FUNCTION_BLOCK "Ponsel_mesure"   // FB107, SCL
{ S7_Optimized_Access := 'TRUE' }
VERSION : 0.1
   VAR_INPUT
      mb_addr : UInt;
      minimum_measurement_interval : Time := T#1M;
      compensate_enable : Bool;
      compensate : Array[1..2] of Real;
   END_VAR
   VAR_OUTPUT
      Measurement_ok : Bool;
   END_VAR
   VAR_IN_OUT
      mb_query : "mb_query";
      start_measurement : Bool;
   END_VAR
   VAR
      sb : "mb_station_block_udt";
      QueryCnt : UDInt;
      data1 : Struct
         value : Array[0..4] of Real;
         compensate_temperature : Real;
         compensate : Array[1..2] of Real;
         _ : Word;
         status : Array[0..4] of Struct
            x08_StmGamme0 : Bool;
            x09_StmGamme1 : Bool;
            x10_StmGamme2 : Bool;
            x11 : Bool;
            x12 : Bool;
            x13 : Bool;
            x14 : Bool;
            x15 : Bool;
            x00_Stm0 : Bool;
            x01_Stm1 : Bool;
            x02_Stm2 : Bool;
            x03_StmTemp : Bool;   // At least one parameter coefficient uses a temporary calibration standard (configuration during calibration)
            x04_StmHF : Bool;   // At least one parameter coefficient is outside calibration limits
            x05_StmCU : Bool;   // All parameter coefficients use default coefficient
            x06_StmHIST : Bool;   // All parameter coefficients use history coefficient
            x07_StmME : Bool;   // Dry weight is missing in at least one parameter coefficient (measurement under way)
         END_STRUCT;
         Compensates_3 : Real;
      END_STRUCT;
      data2 : Struct
         Description : String[30];
         serial_number : String[32];   // (addr 0x0D10)
         Software_version : Word;   // Heavy Weight: Major version and Light Weight: Minor Version.
         Hardware_version : Word;   // Heavy Weight: Major version and Light Weight: Minor Version.
      END_STRUCT;
      api : Struct
         idle : Bool;
         wait : Bool;
         interval : Time;
      END_STRUCT;
      _ : Bool;   // Internal variables bellow.
      state : Int;
      "timer" : TON_TIME;
      timer_in : Bool;
      timer_q : Bool;
      first_scan : Bool := TRUE;
      wait_time : UInt;
   END_VAR
   VAR_TEMP
      "word" : Word;
      c : Int;
      error : Bool;
      tIdle : Bool;
      pt : Time;
   END_VAR
BEGIN
   // Aqualabo - Ponsel mesure
   // Dissolved oxygen (OPTOD), Conductivity (C4E, CTZ), pH_Redox, Turbi    
   // 
   // - Warning: For the oxygen sensor each pull for sensor measurement,
   //   will use of the available life span. Please set the measurement
   //   interval to appropriate value.
   // - Continuous assign true to start_measurement, to continuous do
   //   meassurements. #minimum_measurement_interval wil still restrict
   //   the interval time.
   // - https://en.aqualabo.fr/userfiles/doc/User%20Manual%20Oxygen%20Optical%20digital%20sensor%20OPTOD.pdf

   "mb_station_block_header"(sb := #sb,
                             mb_query := #mb_query);
   #mb_query.mb_addr := #mb_addr;
   #mb_query.mode := #mb_query.c.read.holding_reg;

   #"timer"(IN := #timer_in,
          PT := #"timer".PT,
          Q => #timer_q);
   #timer_in := false;

   IF #sb.out.communication_error THEN // If communication error
       #state := 0;
       #Measurement_ok := false;
       #timer_in := true;  // Continue run the timer.
   ELSE
       CASE #state OF
           1:  // Compensate: Salinity, barometric pressure, temperature, etc.
               IF #compensate_enable THEN
                   #mb_query(mode := #mb_query.c.write.holding_reg,
                             data_addr := 16#5f,
                             data_ptr := #compensate);
                   #state += BOOL_TO_INT(#mb_query.Done);
               ELSE
                   #state += 1;
               END_IF;
           2:  // Read wait-time (Used later in state 4)
               #mb_query(data_addr := 16#A4,
                         data_ptr := #wait_time);
               #state += BOOL_TO_INT(#mb_query.Done);
           3:  // Start all meassurements.
               #"word" := 16#0f;
               #mb_query(mode := #mb_query.c.write.holding_reg,
                         data_addr := 16#01,
                         data_ptr := #"word");
               #state += BOOL_TO_INT(#mb_query.Done);
           4:  // Timer (Wait while sensor is obtaining measurements)
               #timer_in := true;
               PRESET_TIMER(TIMER := #"timer",
                            PT := MAX(IN1 := T_CONV(#wait_time),
                                      IN2 := T#1s)); // No less then 1s.
               #state += BOOL_TO_INT(#timer_q);
           5:  // Get data.
               #mb_query(data_addr := 16#0053,
                         data_ptr := #data1);
               // All measurements ok ?
               FOR #c := 0 TO 4 DO
                   #error := #error
                   OR #data1.status[#c].x00_Stm0
                   OR #data1.status[#c].x01_Stm1
                   OR #data1.status[#c].x02_Stm2;
               END_FOR;
               #Measurement_ok := NOT #error;
               IF #mb_query.Done THEN
                   // #start_measurement need to be assigned
                   // true again to start a new messurement.
                   #start_measurement := false;
                   #state := 0;
                   #QueryCnt += 1;
               END_IF;
           ELSE
               #tIdle := true;
               #timer_in := true;
               #pt := SEL(G := #api.interval = T#0s,
                          IN0 := #api.interval,
                          IN1 := #minimum_measurement_interval);
               PRESET_TIMER(PT := #pt,
                            TIMER := #"timer");

               #state := BOOL_TO_INT
               (NOT #api.wait AND // #api.wait may be set by other
                // function blocks to  halt the messurements.
                #start_measurement AND (
                (* *)#timer_q // Interval controlled
                (* *)OR #first_scan)); // At statup a messurement
               // is done as fast as possible.
       END_CASE;
   END_IF;
   // #wait is a API, for other blocks to stop the messurements,
   // #idle tells other blocks that no messurement is in progress.


   IF #sb.out.communication_error
       OR #api.idle AND NOT #api.wait
   THEN
       // Description, Serial number, sw and hw version.
       #mb_query(data_addr := 3327,
                 data_ptr := #data2);
   END_IF;

   "mb_station_block_footer"(sb := #sb,
                             mb_query := #mb_query);

   #api.idle := #tIdle;
   #api.wait := false;
   #api.interval := T#0s;
   #first_scan := false;

   (* 
   Units:
   ---------------
   value0: Temperature
                         value1:                    value2:                    value3:       
   OPTOD (oxygen)    :   Oxygen [%Sat]              Oxygen [mg/l]              Oxygen [ppm]
   Turbi             :   Nephelo turbidity [NTU]    Nephelo turbidity [FNU]    TU turbidity [mg/L]
   pH_Redox          :   pH                         Redox [mV]
   conductivity_C4E  :   Conductivity C4E [uS/cm]   Salinity [ppt]             TDS - Kcl [ppm]
   Conductivity_CTZ  :   Conductivity CTZ [mS/cm]   Salinity [g/Kg]            Conductivity CTZ [mS/cm] 
                                                                               without temperature compensation                                                                  
   OPTOD: (Dissolved oxygen)
   Compensates[1]: Atmospheric pressure [hPa], default 1013 hPa
   Compensates[2]: Salinity [ppt], default 0 ppt


   Wiring: 
   Red     Wiring diagram V+
   black   Wiring diagram V-
   Green   B+ RS-485  (Siemens A)
   White   A- RS-485  (Siemens B)
   Blue    SDI-12

   Default settings:
   Buad: 9600
   Parity: none
   Modbus address: 10


   StmX:
   000: Measurement OK
   001: Measurement OK, but out of specifications
   010: Measurement OK with INFO 1 (See datasheet)
   011: Measurement OK with INFO 2 (See datasheet)
   100: Measurement impossible, out of specifications
   101: Measurement impossible with INFO 3 (See datasheet)
   110: Measurement impossible with INFO 4 (See datasheet)
   111: measurement under way (not yet available)

   StmGamme:       
   001: measurement used range 1
   010: measurement used range 2
   011: measurement used range 3
   100: measurement used range 4

   *)
END_FUNCTION_BLOCK

// folder: Library/Modbus/Station blocks/sb tested/Siemens

FUNCTION_BLOCK "siemens_PAC3200"   // FB8, SCL
{ S7_Optimized_Access := 'TRUE' }
VERSION : 0.1
   VAR_INPUT
      mb_addr : USInt := 1;
   END_VAR
   VAR_IN_OUT
      mb_query : "mb_query";
   END_VAR
   VAR
      sb : "mb_station_block_udt";
      read1 : Struct
         voltage_L_n : Array[1..3] of Real;
         "voltage _L_L" : Array[1..3] of Real;   // 1:Va-b, 2:Vb-c, 3:Vc-a,
         current : Array[1..3] of Real;
         apparent_power : Array[1..3] of Real;
         active_power : Array[1..3] of Real;
         reactive_power : Array[1..3] of Real;
         power_factor : Array[1..3] of Real;
         THD_R_voltage : Array[1..3] of Real;
      END_STRUCT;
      read2 : Struct
         frequency : Real;   // unit: hz
         avg_voltage_Vph_n : Real;   // unit: V
         avg_voltage_Vph_ph : Real;   // unit: V
         avg_current : Real;   // unit: A
         total_apparent_power : Real;   // unit: VA
         total_active_power : Real;   // unit: W
      END_STRUCT;
   END_VAR
BEGIN
   // Siemens - PAC3200 - Power meter
   // 
   // Manual: 3.9.3, page 40

   "mb_station_block_header"(sb := #sb, mb_query := #mb_query);
   #mb_query.mb_addr := #mb_addr; // Device address.

   // Two queries, reading one section of holding registers each.
   #mb_query.mode := #mb_query.c.read.holding_reg;
   #mb_query(data_addr := 1, data_ptr := #read1);
   #mb_query(data_addr := 55, data_ptr := #read2);
   // - Each query reading one section of holding registers.
   // - Data length is automatically calculated for holding and input regisers.

   "mb_station_block_footer"(sb := #sb, mb_query := #mb_query);
END_FUNCTION_BLOCK

// folder: Library/Modbus/Station blocks/sb tested/zz Internal special

FUNCTION_BLOCK "temeratur_transmitter"   // FB2, SCL
{ S7_Optimized_Access := 'TRUE' }
VERSION : 0.1
   VAR_OUTPUT
      Temperatur : Real;
   END_VAR
   VAR_IN_OUT
      mb_query : "mb_query";
   END_VAR
   VAR
      sb : "mb_station_block_udt";
   END_VAR
   VAR_TEMP
      tmp : Int;
   END_VAR
BEGIN
   // Temperatur transmitter.

   "mb_station_block_header"(sb := #sb, mb_query := #mb_query);

   #mb_query(mb_addr := 1,
             mode := #mb_query.c.read.holding_reg,
             data_addr := 0,
             data_ptr := #tmp);

   IF #mb_query.Done THEN
       #Temperatur := REAL_TO_INT(#tmp) / 10;
   END_IF;

   "mb_station_block_footer"(sb := #sb, mb_query := #mb_query);
END_FUNCTION_BLOCK

// folder: Library/Modbus/Station blocks/sb untested

FUNCTION_BLOCK "Allen_bradley_power_flex_4"   // FB16, SCL
{ S7_Optimized_Access := 'TRUE' }
VERSION : 0.1
   VAR_INPUT
      mb_addr : USInt;
      ref : Real;
      reverse : Bool;
      reset : Bool;
   END_VAR
   VAR_OUTPUT
      Output_Frequency : Real;
      Output_Current : Real;
      DC_Bus_Voltage : Real;
      Output_Voltage : Real;
   END_VAR
   VAR_IN_OUT
      mb_query : "mb_query";
   END_VAR
   VAR
      sb : "mb_station_block_udt";
      read : Struct
         stat : Struct
            x08_At_Reference : Bool;
            x09_Reference_Controlled_by_Comm : Bool;
            x10_Operation_Cmd_Controlled_by_Comm : Bool;
            x11_Parameters_have_been_locked : Bool;
            x12_Digital_Input_1_Status : Bool;
            x13_Digital_Input_2_Status : Bool;
            x14 : Bool;
            x15 : Bool;
            "x00_Ready," : Bool;
            x01_Running : Bool;
            x02_cmd_Forward : Bool;
            x03_Rotating_Forward : Bool;
            x04_Accelerating : Bool;
            "x05_Decelerating," : Bool;
            x06_Alarm : Bool;
            x07_Faulted : Bool;
         END_STRUCT;
         error_code : UInt;
         ref_feedback : UInt;
         Output_Frequency : UInt;
         Output_Current : UInt;
         DC_Bus_Voltage : UInt;
         Output_Voltage : UInt;
      END_STRUCT;
      write : Struct
         cmd : Struct
            "x08_Accel Rate 1" : Bool := TRUE;
            "x09_Accel Rate 2" : Bool;
            "x10_Decel Rate 1" : Bool := TRUE;
            "x11_Decel Rate 2" : Bool;
            x12_Freq_Source_b0 : Bool := TRUE;
            x13_Freq_Source_b1 : Bool := TRUE;
            x14_Freq_Source_b2 : Bool;
            x15 : Bool;
            x00_Stop : Bool;
            x01_Start : Bool;
            x02_Jog : Bool;
            x03_Clear_Faults : Bool;
            x04_Forward : Bool;
            x05_Reverse : Bool;
            x06 : Bool;
            x07 : Bool;
         END_STRUCT;
         ref : UInt;
      END_STRUCT;
   END_VAR
BEGIN
   // Allen Bradley - Power Flex 4 - Compact AC Drive
   //
   // http://ab.rockwellautomation.com/Drives/PowerFlex-4
   // Web: https://plc-hmi-scadas.com/gallery/PowerFlex4ModBusAddressing.pdf

   "mb_station_block_header"(sb := #sb,
                             mb_query := #mb_query);
   #mb_query.mb_addr := #mb_addr;

   #write.ref := REAL_TO_UINT(#ref * 10);
   #write.cmd.x00_Stop := #ref = 0;
   #write.cmd.x01_Start := #ref <> 0;
   #write.cmd.x03_Clear_Faults := #reset;
   #write.cmd.x04_Forward := NOT #reverse;
   #write.cmd.x05_Reverse := #reverse;

   #mb_query.mode := #mb_query.c.write.single_holding_reg;
   #mb_query(data_addr := 8192,
             data_ptr := #write.cmd);
   #mb_query(data_addr := 8193,
             data_ptr := #write.ref);

   #mb_query.mode := #mb_query.c.read.holding_reg;
   #mb_query(data_addr := 8448,
             data_ptr := #read);
   #Output_Frequency := UINT_TO_REAL(#read.Output_Frequency) / 10;
   #Output_Current := UINT_TO_REAL(#read.Output_Current) / 100;
   #DC_Bus_Voltage := UINT_TO_REAL(#read.DC_Bus_Voltage) / 10;
   #Output_Voltage := UINT_TO_REAL(#read.Output_Voltage) / 10;

   "mb_station_block_footer"(sb := #sb,
                             mb_query := #mb_query);

   (* Error codes: (read.error_codes)
   0 - No Fault
   2 - Auxilary Input
   3 - Power Loss
   4 - Undervoltage
   5 - Overvoltage
   6 - Motor Stalled
   7 - Motor Overload
   8 - Heatsink Overtemperature
   12 - HW Overcurrent (300%)
   13 - Ground Fault
   29 - Analog Input Loss
   33 - Auto Restart Tries
   38 - Phase U to Ground Short
   39 - Phase V to Ground Short
   40 - Phase W to Ground Short
   41 - Phase U/V Short
   42 - Phase U/W Short
   43 - Phase V/W Short
   63 - Software Overcurrent
   64 - Drive Overload
   70 - Power Unit Fail
   80 - AutoTune Fail
   81 - Communication Loss
   100 - Parameter Checksum Error
   122 - I/O Board Fail         
   *)
END_FUNCTION_BLOCK

FUNCTION_BLOCK "Auma_valve"   // FB17, SCL
{ S7_Optimized_Access := 'TRUE' }
VERSION : 0.1
   VAR_INPUT
      mb_addr : UInt;
   END_VAR
   VAR_IN_OUT
      mb_query : "mb_query";
   END_VAR
   VAR
      sb : "mb_station_block_udt";
      read : Struct
         status : Struct
            torque_sw_closed : Bool;
            torque_sw_open : Bool;
            limit_sw_closed : Bool;
            limit_sw_open : Bool;
            sel_sw_local : Bool;
            sel_sw_remote : Bool;
            phase_fault : Bool;
            therminal_fault : Bool;
            falt : Bool;
            warning : Bool;
            running_close : Bool;
            running_open : Bool;
            not_ready_remote : Bool;
            setpoint_reached : Bool;
            end_p_clossed : Bool;
            end_p_open : Bool;
         END_STRUCT;
         "Actual position" : UInt;
      END_STRUCT;
      write : Struct
         cmd : Struct
            byte_2 : Byte;
            open : Bool;
            close : Bool;
            use_setpoint : Bool;
            reset : Bool;
            b4 : Bool;
            b5 : Bool;
            b6 : Bool;
            b7 : Bool;
         END_STRUCT;
         setpoint : UInt;
      END_STRUCT;
   END_VAR
BEGIN
   // Auma actuator controls
   // AC 01.2/ACExC 01.2 Modbus RTU
   //
   // http://www1.auma.com/uploads/media/sp_import2/handbuecher/
   // steuerungen/hb_ac2_modbus_geraeteintegration_en.pdf

   "mb_station_block_header"(sb := #sb, mb_query := #mb_query);
   #mb_query.mb_addr := #mb_addr;

   #mb_query(mode := #mb_query.c.read.input_reg,
             data_addr := 16#03E8,
             data_ptr := #read); // p.10

   #mb_query(mode := #mb_query.c.write.holding_reg,
             data_addr := 16#03E8,
             data_ptr := #write); // p.29

   "mb_station_block_footer"(sb := #sb, mb_query := #mb_query);

   (*
   - Each query reading one section of holding registers.
   - Data length is automatically calculated for holding 
     and input regisers.
   *)
END_FUNCTION_BLOCK

FUNCTION_BLOCK "Automatic_systems_AS1320"   // FB18, SCL
{ S7_Optimized_Access := 'TRUE' }
VERSION : 0.1
   VAR_INPUT
      mb_addr : UInt;
   END_VAR
   VAR_IN_OUT
      mb_query : "mb_query";
   END_VAR
   VAR
      sb : "mb_station_block_udt";
      read1 : Struct
         input : Word;
         input_3 : Word;
         output : Word;
         analog_in : Word;
         analog_out : Word;
         z2 : Array[1..4] of Word;
         temperature : Int;
         counter_1 : UDInt;
         counter_2 : UDInt;
         z : Array[1..3] of Word;
         state : Struct
            x08_blocked_closed : Bool;
            x09 : Bool;
            x10 : Bool;
            x11 : Bool;
            x12 : Bool;
            x13 : Bool;
            x14 : Bool;
            x15 : Bool;
            x00 : Bool;
            x01 : Bool;
            x02_open : Bool;
            x03_opening : Bool;
            x04_closed : Bool;
            x05_closing : Bool;
            x06_stop : Bool;
            x07_blocked_open : Bool;
         END_STRUCT;
      END_STRUCT;
      read2 : Struct
         PRDSTD : String[6];
         BL_xxx : String[6];
         "Type" : UInt;
         Change : UInt;
      END_STRUCT;
      write1 : Struct
         x08 : Bool;
         x09 : Bool;
         x10 : Bool;
         x11 : Bool;
         x12 : Bool;
         x13 : Bool;
         x14 : Bool;
         x15 : Bool;
         x00_open : Bool;
         x01_close : Bool;
         x02_block_open : Bool;
         x03_block_close : Bool;
         x04_stop : Bool;
         x05_reader_command_direction_a : Bool;
         x06_reader_command_direction_b : Bool;
         x07_reset_block : Bool;
      END_STRUCT;
      start_setup : Bool;
      write2 : Struct
         PS1_function : UInt;
         PS2_function : UInt;
         Positioning : UInt;
         barrier_type : UInt;
         arm_length : UInt;
         arm_type : UInt;
         power_fail_OP : UInt;
         exploitation : UInt;
      END_STRUCT;
      crank : Bool;
   END_VAR
BEGIN
   // Automatic systems - AS1320
   // http://www.visionbr.com.br/arquivo-produtos/20110823_92924_as1320-mt-en-16.pdf
   // Revision no: AS1320-prog 6.x-MT-FR-16 - 2009-11-10 

   "mb_station_block_header"(sb := #sb, mb_query := #mb_query);
   #mb_query.mb_addr := #mb_addr;

   #mb_query.mode := #mb_query.c.read.holding_reg;
   #mb_query(data_addr := 16#39, data_ptr := #read1);
   // #mb_query(data_addr := 16#00, data_ptr := #read3);
   // A micro switch at opening for the crank.
   #crank := #read1.input.%X14; 

   #mb_query.mode := #mb_query.c.write.holding_reg;
   #mb_query(data_addr := 16#12C, data_ptr := #write1);
   IF #start_setup THEN
       #mb_query(data_addr := 16#64, data_ptr := #write2);
       #start_setup := NOT #mb_query.Done;
   END_IF;

   "mb_station_block_footer"(sb := #sb, mb_query := #mb_query);
END_FUNCTION_BLOCK

FUNCTION_BLOCK "Belimo_vav_Compact_mod"   // FB19, SCL
{ S7_Optimized_Access := 'TRUE' }
VERSION : 0.1
   VAR_INPUT
      mb_addr : UInt;
      sp : Real;   // setpoint
      bus_fail_position : Real;
   END_VAR
   VAR_OUTPUT
      pos_feedback : Real;
   END_VAR
   VAR_IN_OUT
      mb_query : "mb_query";
   END_VAR
   VAR
      sb : "mb_station_block_udt";
      read : Struct
         position : Int;
      END_STRUCT;
      write1 : Struct
         setpoint : Int;
      END_STRUCT;
      write2 : Struct
         bus_fail_position : Int;
      END_STRUCT;
   END_VAR
BEGIN
   // Belimo - VAV-Compact MOD 
   // LMV-D3-MOD 5  Nm 2   W 4 VA (max. 5 A @ 5 ms) Approx. 500 g
   // NMV-D3-MOD 10 Nm 3.5 W 6 VA (max. 5 A @ 5 ms) Approx. 700 g
   // https://www.micromatic.no/globalassets/inriver/
   // resources/ko1070_0_5_1.pdf

   "mb_station_block_header"(sb := #sb, mb_query := #mb_query);
   #mb_query.mb_addr := #mb_addr;

   #mb_query.mode := #mb_query.c.read.holding_reg;
   #mb_query(data_addr := 4, data_ptr := #read);
   #pos_feedback := INT_TO_REAL(#read.position) * 0.01;

   #mb_query.mode := #mb_query.c.write.holding_reg;
   #write1.setpoint := REAL_TO_INT(#sp) * 100;
   #mb_query(data_addr := 0, data_ptr := #write1);
   #write2.bus_fail_position := REAL_TO_INT(#bus_fail_position) * 100;
   #mb_query(data_addr := 108, data_ptr := #write2);

   "mb_station_block_footer"(sb := #sb, mb_query := #mb_query);

   (*
   Bus fail position:
   0 Last setpoint (no bus monitoring)
   1 Fast close if time is exceeded
   2 Fast open if time is exceeded 
   *)
END_FUNCTION_BLOCK

FUNCTION_BLOCK "Binmaster_mnu_ultrasonic_sensor"   // FB20, SCL
{ S7_Optimized_Access := 'TRUE' }
VERSION : 0.1
   VAR_INPUT
      mb_addr : UInt;
   END_VAR
   VAR_IN_OUT
      mb_query : "mb_query";
   END_VAR
   VAR
      sb : "mb_station_block_udt";
      data : Struct
         "Model Type" : UInt;
         Raw_Distance_Level : UInt;   // [mm]
         _ : UInt;
         Temperature : Int;
         Calculated : DInt;
         __ : DWord;
         "Version" : UInt;
         "Signal Strength" : UInt;
         ___ : UInt;
         "Trip 1 Alarm" : UInt;
         "Trip 1 Status" : UInt;
         "Trip 2 Alarm" : UInt;
         "Trip 2 Status" : UInt;
      END_STRUCT;
      setting : Struct
         Units : UInt := 3;   // 3=Meters
         Distance : Struct
            Max : UInt;   // 0 - 15,250 mm
            Full : UInt;   // 0 - 15,250 mm
            Empty : UInt;
         END_STRUCT;
         cal : Struct
            Multiplier : UInt := 1000;   // 1000 -> 1.000
            Offset : UInt := 0;
         END_STRUCT;
      END_STRUCT;
   END_VAR
BEGIN
   // Binmaster - MNU Ultrasonic Sensor
   // 
   // Web: http://www.binmaster.com/_resources/e30d:ogspbx-on/files/
   // 75651567z4d4b98f5/_fn/BinMaster%20MNU%20manual%209004257%20Rev%20A1.pdf

   "mb_station_block_header"(sb := #sb, mb_query := #mb_query);
   #mb_query.mb_addr := #mb_addr;

   #mb_query.mode := #mb_query.c.mode.read;
   #mb_query(data_addr := 30299, data_ptr := #data);

   #mb_query.mode := #mb_query.c.mode.write;
   #mb_query(data_addr := 40401, data_ptr := #setting.Units);
   #mb_query(data_addr := 40405, data_ptr := #setting.Distance);
   #mb_query(data_addr := 40416, data_ptr := #setting.cal);

   "mb_station_block_footer"(sb := #sb, mb_query := #mb_query);
END_FUNCTION_BLOCK

FUNCTION_BLOCK "Delta_CFP2000"   // FB22, SCL
{ S7_Optimized_Access := 'TRUE' }
VERSION : 0.1
   VAR_INPUT
      mb_addr : USInt;
      ref : Real;   // (minus=>rev.)
   END_VAR
   VAR_OUTPUT
      stat : Struct
         drive_stops : Bool;
         drive_decelerating : Bool;
         drive_standby : Bool;
         drive_operating : Bool;
      END_STRUCT;
      current : Real;
   END_VAR
   VAR_IN_OUT
      mb_query : "mb_query";
   END_VAR
   VAR
      sb : "mb_station_block_udt";
      read : Struct
         warn_code : USInt;
         error_code : USInt;
         stat : Struct
            "b08_Master frequency controlled by communication" : Bool;
            "b09 Master frequency controlled by analog signal" : Bool;
            "b10 Operation command controlled by communication interface" : Bool;
            "b11 Parameter locked" : Bool;
            "b12 Enable to copy parameters from keypad" : Bool;
            b13 : Bool;
            b14 : Bool;
            b15 : Bool;
            b00_oper_stat : Bool;
            b01_oper_stat : Bool;
            b02 : Bool;
            b03_direction : Bool;
            b04_direction : Bool;
            b05 : Bool;
            b06 : Bool;
            b07 : Bool;
         END_STRUCT;
         frequency_cmd : Int;
         output_frequency : Int;
         output_current : UInt;
         "DC-BUS Voltage" : UInt;
         output_voltage : UInt;
         "Current step number of Multi-Step Speed Operation" : Int;
         _ : Int;
         counter_value : Int;
         power_factor_angle : Int;
         output_torque : Int;
         actual_motor_speed : Int;
         __ : Int;
         ___ : Int;
         power_output : Int;   // kwh
      END_STRUCT;
      write : Struct
         cmd_word : Struct
            b08_sel_speed : Bool;
            b09_sel_speed : Bool;
            b10_sel_speed : Bool;
            b11_sel_speed : Bool;
            b12_Enable_bit06_11_function : Bool := TRUE;
            b13_oper_keypad : Bool;
            b14_oper_Pr_00_21_setting : Bool;
            b15 : Bool;
            b00_stop : Bool;
            b01_run : Bool;
            b02 : Bool;
            b03 : Bool;
            b04_fwd : Bool;
            b05_rev : Bool;
            b06_sel_accel_decel : Bool;
            b07_sel_accel_decel : Bool;
         END_STRUCT;
         ref_freq : UInt;
         "a" : Struct
            b08 : Bool;
            b09 : Bool;
            b10 : Bool;
            b11 : Bool;
            b12 : Bool;
            b13 : Bool;
            b14 : Bool;
            b15 : Bool;
            b00_external_fault : Bool;
            b01_reset : Bool;
            b02_B_B_ON : Bool;
            b03 : Bool;
            b04 : Bool;
            b05 : Bool;
            b06 : Bool;
            b07 : Bool;
         END_STRUCT;
      END_STRUCT;
   END_VAR
BEGIN
   // Delta - CFP2000 - Variable frequency drive
   // 
   // http://www.softstartuk.com/wp-content/uploads/2017/07/VFD-CFP2000_UM_EN_20170303.pdf

   "mb_station_block_header"(sb := #sb, mb_query := #mb_query);
   #mb_query.mb_addr := #mb_addr;

   // Read
   #mb_query.mode := #mb_query.c.read.holding_reg;

   #mb_query(data_addr := 16#2100, data_ptr := #read);
   #stat.drive_stops := NOT #read.stat.b00_oper_stat AND NOT #read.stat.b01_oper_stat;
   #stat.drive_decelerating := #read.stat.b00_oper_stat AND NOT #read.stat.b01_oper_stat;
   #stat.drive_standby := NOT #read.stat.b00_oper_stat AND #read.stat.b01_oper_stat;
   #stat.drive_operating := #read.stat.b00_oper_stat AND #read.stat.b01_oper_stat;
   #current := UINT_TO_REAL(#read.output_current) * 100;
   // Output current (XX.XX A). When current is higher than
   // 655.35, it will shift decimal as (XXX.XA). The decimal
   // can refer to High byte of 211F. 

   // Write
   #mb_query.mode := #mb_query.c.write.holding_reg;

   #write.ref_freq := REAL_TO_UINT(#ref * 100);
   #write.cmd_word.b00_stop := #ref = 0;
   #write.cmd_word.b01_run := NOT #write.cmd_word.b00_stop;
   #write.cmd_word.b05_rev := #ref < 0;
   #write.cmd_word.b04_fwd := NOT #write.cmd_word.b05_rev;
   #mb_query(data_addr := 16#2000, data_ptr := #write);

   "mb_station_block_footer"(sb := #sb, mb_query := #mb_query);
END_FUNCTION_BLOCK

FUNCTION_BLOCK "Emerson_Micro_Motion"   // FB23, SCL
{ S7_Optimized_Access := 'TRUE' }
VERSION : 0.1
   VAR_INPUT
      mb_addr : UInt;
   END_VAR
   VAR_IN_OUT
      mb_query : "mb_query";
   END_VAR
   VAR
      sb : "mb_station_block_udt";
      data : Struct
         stat : Struct
            x08_Primary_mA_output_saturated : Bool;
            x09_Secondary_mA_output_saturated : Bool;
            x10_Primary_mA_output_fixed : Bool;
            x11_Secondary_mA_output_fixed : Bool;
            x12_Density_overrange : Bool;
            x13_Flowmeter_zeroing_failure : Bool;
            x14_Zero_value_too_low : Bool;
            x15_Zero_value_too_high : Bool;
            x00_EPROM_checksum_failure : Bool;
            x01_RAM_diagnostic_failure : Bool;
            x02_Sensor_failure : Bool;
            x03_Temperature_sensor_failure : Bool;
            x04_Input_overrange : Bool;
            x05_Frequency_pulse_output_saturated : Bool;
            x06_Transmitter_not_configured : Bool;
            x07_Realtime_interrupt_failure : Bool;
            x24 : Bool;
            x25 : Bool;
            x26 : Bool;
            x27 : Bool;
            x28 : Bool;
            x29 : Bool;
            x30 : Bool;
            x31 : Bool;
            x16_Transmitter_electronics_failure : Bool;
            x17_Flowmeter_zeroing_in_progress : Bool;
            x18_Slug_flow : Bool;
            x19_Power_reset_occurred : Bool;
            x20_Transmitter_configuration_changed : Bool;
            x21_Transmitter_initializing_warming_up : Bool;
            x22 : Bool;
            x23 : Bool;
         END_STRUCT;
         "Mass flow rate" : Real;
         Density : Real;
         Temperature : Real;
         "Volume flow rate" : Real;
         Pressure : Real;   // (internally derived)
         "Mass total" : Real;
         "Volume total" : Real;
         "Mass inventory" : Real;
         "Volume inventory" : Real;
      END_STRUCT;
   END_VAR
BEGIN
   // Emerson - Micro Motion Transmitters
   // RFT9739, MVD DC, Modeo 1500, Model 1700, Model 2500, Model 2700, Series 3000
   // 
   // Web: http://www2.emersonprocess.com/siteadmincenter/
   //      PM%20Micro%20Motion%20Documents/Modbus-Map-Manual-20001741.pdf

   "mb_station_block_header"(sb := #sb, mb_query := #mb_query);
   #mb_query.mb_addr := #mb_addr;

   #mb_query.mode := #mb_query.c.read.holding_reg;
   #mb_query(data_addr := 245, data_ptr := #data);

   "mb_station_block_footer"(sb := #sb, mb_query := #mb_query);
END_FUNCTION_BLOCK

FUNCTION_BLOCK "Endress_proline_promass_83"   // FB24, SCL
{ S7_Optimized_Access := 'TRUE' }
VERSION : 0.1
   VAR_INPUT
      mb_addr : UInt;
   END_VAR
   VAR_OUTPUT
      device_ok : Bool;
   END_VAR
   VAR_IN_OUT
      mb_query : "mb_query";
   END_VAR
   VAR
      sb : "mb_station_block_udt";
      data : Struct
         mass_flow : Real;
         temperature : Real;
         totalizer : Real;
         actual_system_condition : Int;   // 1->ok
      END_STRUCT;
   END_VAR
BEGIN
   // Endress - Proline Promass 83
   // Web: https://portal.endress.com/wa001/dla/5000000/5862/000/05/BA00107DEN_1311.pdf

   "mb_station_block_header"(sb := #sb, mb_query := #mb_query);
   #mb_query.mb_addr := #mb_addr;

   #mb_query(mode := #mb_query.c.read.holding_reg,
             data_addr := 5051,
             data_ptr := #data);

   "mb_station_block_footer"(sb := #sb, mb_query := #mb_query);

   #device_ok := #data.actual_system_condition = 1;
END_FUNCTION_BLOCK

FUNCTION_BLOCK "Epluse_EE071"   // FB25, SCL
{ S7_Optimized_Access := 'TRUE' }
VERSION : 0.1
   VAR_INPUT
      mb_addr : USInt := 247;
   END_VAR
   VAR_IN_OUT
      mb_query : "mb_query";
   END_VAR
   VAR
      sb : "mb_station_block_udt";
      data : Struct
         temperature_C : Real;   // [Â°C]
         temperature_F : Real;   // [Â°F]
         humidity_rel : Real;   // [%]
         humidity_abs : Real;   // [g/mÂ³]
      END_STRUCT;
      serial : String[8];
   END_VAR
BEGIN
   // Epluse - EE071
   // Humidity and Temperature Probe
   //
   // http://downloads.epluse.com/fileadmin/data/product/ee071/datasheet_EE071.pdf

   "mb_station_block_header"(sb := #sb,
                             mb_query := #mb_query);
   #mb_query.mb_addr := #mb_addr;

   #mb_query.mode := #mb_query.c.read.holding_reg;
   #mb_query(data_addr := 30026,
             data_ptr := #data);
   #mb_query(data_addr := 30001,
             data_ptr := #serial); // 30001-30008

   "mb_station_block_footer"(sb := #sb,
                             mb_query := #mb_query);

   IF #sb.out.communication_error THEN
       #data.temperature_C := 0;
       #data.temperature_F := 0;
       #data.humidity_rel := 0;
       #data.humidity_abs := 0;
   END_IF;

   (* Electrical connections

   Supply voltage 1) 2) 4 - 28 V DC

   brown...+UB
   white.....B-RS485 (= Data-)
   blue......A-RS485 (= Data+)
   black....GND
   grey......shielding

   1...+UB
   2...B-RS485 (= Data-)
   3...A-RS485 (= Data+)
   4...GND

   *)
END_FUNCTION_BLOCK

FUNCTION_BLOCK "G_Instruments_GpH141_MB"   // FB26, SCL
{ S7_Optimized_Access := 'TRUE' }
VERSION : 0.1
   VAR_INPUT
      mb_addr : USInt;
   END_VAR
   VAR_OUTPUT
      voltage_mV : Real;
      pH : Real;
      temperature : Real;
   END_VAR
   VAR_IN_OUT
      mb_query : "mb_query";
   END_VAR
   VAR
      sb : "mb_station_block_udt";
      change_mb_addr : Struct
         old : UInt;
         new : UInt;
      END_STRUCT;
   END_VAR
   VAR_TEMP
      read1 : Struct
         voltage : Int;
         pH : Int;   // compensated for temperature
         temperature : Int;
      END_STRUCT;
   END_VAR
BEGIN
   // G Instruments - GpH141-MB - pH/ORP Transmitter
   // Part number: 30535.
   // http://www.ginstruments.com/files/GpH141-MB.pdf

   "mb_station_block_header"(sb := #sb,
                             mb_query := #mb_query);
   #mb_query.mb_addr := #mb_addr;

   #mb_query.mode := #mb_query.c.read.holding_reg;

   #mb_query(data_addr := 19,
             data_ptr := #read1);
   IF #mb_query.Done THEN
       #voltage_mV := INT_TO_REAL(#read1.voltage) / 10;
       #pH := INT_TO_REAL(#read1.pH) / 100;
       #temperature := INT_TO_REAL(#read1.temperature) / 10;
   END_IF;

   (* IF #change_mb_addr.new <> 0 AND #change_mb_addr.old <> 0 THEN
       #mb_query(mb_addr := #change_mb_addr.old,
                 mode := #mb_query.c.write.single_holding_reg,
                 data_addr := 1200,
                 data_ptr := #change_mb_addr.new);
       IF #mb_query.Done THEN #change_mb_addr.new := 0; END_IF;
   END_IF; *)

   "mb_station_block_footer"(sb := #sb,
                             mb_query := #mb_query);

   (*
   Default comm. setting: 19200 bps, even parity, addr 1.

   Electrical connection:
   10 is A (D+)
   11 is RS485 ground (isolated from all other grounds)
   12 is B (D-)
   *)
END_FUNCTION_BLOCK

FUNCTION_BLOCK "hitachi_wj200_series"   // FB27, SCL
{ S7_Optimized_Access := 'TRUE' }
VERSION : 0.1
   VAR_INPUT
      mb_addr : USInt;
      ref : Real;
      acceleration_time : Real := 30.0;   // sec
      deceleration_time : Real := 30.0;   // sec
   END_VAR
   VAR_OUTPUT
      output_frequency : Real;
      output_current : Real;
   END_VAR
   VAR_IN_OUT
      mb_query : "mb_query";
   END_VAR
   VAR
      sb : "mb_station_block_udt";
      save_param : Bool;
      read1 : Struct
         output_frequency : UDInt;   // 0.01 [Hz]
         output_current : UInt;   // 0.1 [A]
         rotation_direction : Int;   // 0: Stopping, 1: Forward, 2:Reverse
      END_STRUCT;
      read2 : Struct
         torque : Int;   // [%]
         output_voltage : UInt;   // 0.1 [V]
         output_power : UInt;   // 0.1 [kW]
         watt_hour : UDInt;   // 0.1 [wh]
         elapsed_run_time : UDInt;   // [h]
         elapsed_power_on_time : UDInt;   // [h]
         "heat sink_temperature" : UDInt;   // 0.1 [℃]
      END_STRUCT;
      read3_Life_check : Struct
         x08 : Bool;
         x09 : Bool;
         x10 : Bool;
         x11 : Bool;
         x12 : Bool;
         x13 : Bool;
         x14 : Bool;
         x15 : Bool;
         x00_Capacitor_on_main_circuit_board : Bool;
         x01_cooling_fan : Bool;
         x02 : Bool;
         x03 : Bool;
         x04 : Bool;
         x05 : Bool;
         x06 : Bool;
         x07 : Bool;
      END_STRUCT;
      read4_Ambient_temperature : Int;
      read5_trip : Struct
         cnt : UInt;
         info : Array[1..3] of Struct
            factor : UInt;
            status : UInt;
            frequency : DInt;
            current : UInt;
            voltage : UInt;
            running_time : UDInt;   // [h] Cumulative running time at tripping
            powerOn_time : UDInt;   // [h] Cumulative power-on time at tripping
         END_STRUCT;
      END_STRUCT;
      read6_status : Struct
         "A" : UInt;
         "B" : UInt;   // 0: Stopping, 1: Running, 2: Tripping
         C : UInt;
      END_STRUCT;
      read7 : Struct
         x0_inverter_ready : Bool;
         x1_forward : Bool;
         x2_reverse : Bool;
         x3_major_failure : Bool;
         x4_data_writing_in_progress : Bool;
         x5 : Bool;
         x6 : Bool;
         x7 : Bool;
      END_STRUCT;
      write1 : Struct
         acceleration_time_1 : UDInt := 3000;   // x0.01 sec
         deceleration_time_1 : UDInt := 3000;   // x0.01 sec
      END_STRUCT;
      write2_source : Struct
         frequency_source : UInt := 3;   // 3:Modbus
         run_command_source : UInt := 3;   // 3:Modbus
      END_STRUCT;
      write3_comm_error : Struct
         communication_watchdog_timer : UInt := 1000;   // 0.01 [sec.]
         communication_error_action : UInt := 4;
      END_STRUCT;
      write5 : Struct
         x0_Run : Bool;
         x1_Reverse : Bool;
         x2_Trip : Bool;
         x3_Reset : Bool;
         x4 : Bool;
         x5 : Bool;
         x6 : Bool;
         x7 : Bool;
      END_STRUCT;
      write6_DC_breaking : Struct
         enable : UInt;   // 0 (disabling), 1 (enabling), 2 (output freq < [A052])
         frequency : UInt;   // 0.01 [Hz]
         wait_time : UInt;   // 0.1 [sec.]
         force_during_deceleration : UInt;   // [%]
         time_for_deceleration : UInt;   // 0.1 [sec.]
      END_STRUCT;
   END_VAR
   VAR_TEMP
      tmp : Word;
      write4_frequency : DInt;   // 0.01 [Hz]
   END_VAR
BEGIN
   // Hitachi WJ200-series
   // Manual Number: NT325X
   // https://www.hitachi-america.us/supportingdocs/forbus/inverters/Support/WJ200_Instruction_NT325X.pdf

   "mb_station_block_header"(sb := #sb, mb_query := #mb_query);
   #mb_query.mb_addr := #mb_addr;

   // --- Read queries
   #mb_query.mode := #mb_query.c.read.holding_reg;
   #mb_query(data_addr := 16#1001, data_ptr := #read1);
   #mb_query(data_addr := 16#1010, data_ptr := #read2);
   #mb_query(data_addr := 16#101d, data_ptr := #read3_Life_check);
   #mb_query(data_addr := 16#134e, data_ptr := #read4_Ambient_temperature);
   #mb_query(data_addr := 16#0011, data_ptr := #read5_trip);
   #mb_query(data_addr := 16#0003, data_ptr := #read6_status);

   #output_frequency := UDINT_TO_REAL(#read1.output_frequency) / 100;
   #output_current := UINT_TO_REAL(#read1.output_current) / 10;

   #mb_query(mode := #mb_query.c.read.discrete_output,
             data_addr := 16#0045,
             data_ptr := #read7);

   // --- Write queries ---
   #write4_frequency := REAL_TO_DINT(#ref * 100);
   #write1.acceleration_time_1 := REAL_TO_UDINT(#acceleration_time * 100);
   #write1.deceleration_time_1 := REAL_TO_UDINT(#deceleration_time * 100);

   #mb_query.mode := #mb_query.c.write.holding_reg;
   #mb_query(data_addr := 16#1103, data_ptr := #write1);
   #mb_query(data_addr := 16#1201, data_ptr := #write2_source);
   #mb_query(data_addr := 16#162e, data_ptr := #write3_comm_error);
   #mb_query(data_addr := 16#0001, data_ptr := #write4_frequency);
   #mb_query(data_addr := 16#1245, data_ptr := #write6_DC_breaking);

   // Save data to EEPROM. 
   IF #save_param THEN
       #mb_query(mode := #mb_query.c.write.single_holding_reg,
                 data_addr := 16#0900,
                 data_ptr := #tmp);
       #save_param := NOT #mb_query.Done;
   END_IF;

   #write5.x0_Run := #ref <> 0;
   #mb_query(mode := #mb_query.c.write.discrete_output,
             data_addr := 16#0001,
             data_len := 4,
             data_ptr := #write5);

   #mb_query.data_len := #mb_query.c.auto_len;
   "mb_station_block_footer"(sb := #sb, mb_query := #mb_query);

   (*
   === read6_status ===
   .A
   0: Initial status
   2: Stopping
   3: Running
   4: Free-run stop
   5: Jogging
   6: DC braking
   7: Retrying
   8: Tripping
   9: Undervoltage (UV), 

   .C
   1: Stopping
   2: Decelerating
   3: Constant-speed operation
   4: Accelerating
   5: Forward rotation
   6: Reverse rotation
   7: Switching from fwd. to rev. rotation,
   8: Switching from rev. to fwd. rotation,
   9: Starting fwd.
   10: Starting rev

   === write3_comm_error.communication_error_action === 
   0 (tripping), 
   1 (tripping after decelerating and stopping the motor), 
   2 (ignoring errors),
   3 (stopping the motor after free-running),
   4 (decelerating and stopping the motor) 

   === Save data to EEPROM === 
   The service life of the storage element of the inverter is 
   limited to about 100,000 write operations.  Frequent use of 
   the ENTER command may shorten its service life.

   === read5_trip.info ===
   .factor: 
   00 No trip factor 0 
   01 Over-current event while at constant speed 1 
   02 Over-current event during deceleration 2 
   03 Over-current event during acceleration 3 
   04 Over-current event during other conditions 4 
   05 Overload protection 5 
   06 Braking resistor overload protection 6 
   07 Overvoltage protection 7 
   08 EEPROM error 8 
   09 Undervoltage protection 9
   10 Current detection error 10
   11 CPU error 11
   12 External trip 12
   13 USP error 13
   14 Ground-fault protection 14
   15 Input overvoltage protection 15
   21 Inverter thermal trip 21
   22 CPU error 22
   25 Main circuit error 25
   30 Driver error 30
   35 Thermistor error 35
   36 Braking error 36
   37 Safe Stop 37
   38 Low-speed overload protection 38
   40 Operator connection 40
   41 Modbus communication error 41
   43 Easy sequence error (invalid instruction) 43
   44 Easy sequence error (invalid nesting count) 44
   45 Easy sequence execution error 1 45
   50 Easy sequence user trip 0 to 9, 50 to 59
   60 Option error 0 to 9, 60 to 69
   80 Encoder disconnection 80
   81 Excessive speed 81
   83 Position control range trip 83

   .status
   0: Resetting 
   1: Stopping 
   2: Decelerating 
   3: Constant-speed operation 
   4: Accelerating 
   5: Operating at zero frequency 
   6: Starting 
   7: DC braking 
   8: Overload restricted 

   *)
END_FUNCTION_BLOCK

FUNCTION_BLOCK "InSitu_RDO_PRO_X"   // FB30, SCL
{ S7_Optimized_Access := 'TRUE' }
VERSION : 0.1
   VAR_INPUT
      mb_addr : UInt;
   END_VAR
   VAR_OUTPUT
      dissolved_oxygen : Real;   // mg/L
      temperature : Real;   // C
      saturation : Real;   // %
      oxygen_partial_pressure : Real;   // mbar
      alarm : Bool;
   END_VAR
   VAR_IN_OUT
      mb_query : "mb_query";
   END_VAR
   VAR
      sb : "mb_station_block_udt";
      read1 : Array[1..4] of Struct
         value : Real;
         Parameter_ID : UInt;
         Units_ID : UInt;
         data_quality : UInt;
         "Off line_sentinel_value" : UInt;
         Available_Units : UInt;
      END_STRUCT;
      read2 : Struct
         serial_number : UDInt;
         manufacture_date : Array[1..3] of UInt;
      END_STRUCT;
      device_name : String[32];
   END_VAR
   VAR_TEMP
      tmp_alarm : Bool;
      c : Int;
   END_VAR
BEGIN
   // InSitu - RDO PRO X
   // 
   // https://in-situ.com/wp-content/uploads/2015/08/
   // RDO_PRO-X_-Titan_Modbus_SDI-12-_Guide.pdf

   "mb_station_block_header"(sb := #sb, mb_query := #mb_query);
   #mb_query.mb_addr := #mb_addr;

   #mb_query.mode := #mb_query.c.read.holding_reg;
   #mb_query(data_addr := 38, data_ptr := #read1);
   #mb_query(data_addr := 9002, data_ptr := #read2);
   #mb_query(data_addr := 9019, data_ptr := #device_name);

   #dissolved_oxygen := #read1[1].value;
   #temperature := #read1[2].value;
   #saturation := #read1[3].value;
   #oxygen_partial_pressure := #read1[4].value;
   FOR #c := 1 TO 4 DO
       #tmp_alarm := #tmp_alarm OR #read1[#c].data_quality <> 0;
   END_FOR;
   #alarm := #tmp_alarm;

   "mb_station_block_footer"(sb := #sb, mb_query := #mb_query);

   (* 
   === Sensor health table: ===
   0  Normal Data Quality
   1  Parameter measured without errors using an expired user 
      calibration. (User Cal Expired)
   2  Parameter measured without errors using an expired factory 
      calibration. (Factory Cal Expired)
   3  Parameter measured with error, sentinel value supplied. 
   4  Sensor is warming up, sentinel value supplied.
   5  Parameter measured but does not meet normal quality 
      criteria. The sensor has sustained moderate damage, or  
      the recommended lifespan has been reached.
   *)
END_FUNCTION_BLOCK

FUNCTION_BLOCK "Jdrk_RS_WS_N01_8"   // FB31, SCL
{ S7_Optimized_Access := 'TRUE' }
VERSION : 0.1
   VAR_OUTPUT
      Temperature : Real;
   END_VAR
   VAR_IN_OUT
      mb_query : "mb_query";
   END_VAR
   VAR
      sb : "mb_station_block_udt";
   END_VAR
   VAR RETAIN
      offset : Real;
   END_VAR
   VAR_TEMP
      tmp : Int;
   END_VAR
BEGIN
   // JDRK - RS-WS-N01-8 - Temperature and Humidity sensor

   "mb_station_block_header"(sb := #sb, mb_query := #mb_query);

   #mb_query(mb_addr := 1,
             mode := #mb_query.c.read.input_reg,
             data_addr := 1,
             data_ptr := #tmp);

   IF #mb_query.Done THEN
       #Temperature := INT_TO_REAL(#tmp) / 10 + #offset;
   END_IF;

   "mb_station_block_footer"(sb := #sb, mb_query := #mb_query);
END_FUNCTION_BLOCK

FUNCTION_BLOCK "Moxa_ioLogik_R1200"   // FB36, SCL
{ S7_Optimized_Access := 'TRUE' }
VERSION : 0.1
   VAR_INPUT
      mb_addr : UInt;
   END_VAR
   VAR_IN_OUT
      mb_query : "mb_query";
   END_VAR
   VAR
      sb : "mb_station_block_udt";
      in : Array[0..15] of Bool;
      out : Array[0..15] of Bool;
   END_VAR
BEGIN
   // Moxa - ioLogik R1200
   // 
   // Web: https://www.moxa.com/doc/man/ioLogik_R1200_Series_UM_e3.1.pdf

   "mb_station_block_header"(sb := #sb,
                             mb_query := #mb_query);
   #mb_query.mb_addr := #mb_addr;

   #mb_query(mode := #mb_query.c.read.discrete_input,
             data_addr := 0,
             data_ptr := #in);

   #mb_query(mode := #mb_query.c.write.discrete_output,
             data_addr := 16#140,
             data_ptr := #out);

   "mb_station_block_footer"(sb := #sb,
                             mb_query := #mb_query);
END_FUNCTION_BLOCK

FUNCTION_BLOCK "MTS_sensors_M_Series"   // FB37, SCL
{ S7_Optimized_Access := 'TRUE' }
VERSION : 0.1
   VAR_INPUT
      mb_addr : UInt;
   END_VAR
   VAR_OUTPUT
      level : Real;
      temperature : Real;
   END_VAR
   VAR_IN_OUT
      mb_query : "mb_query";
   END_VAR
   VAR
      sb : "mb_station_block_udt";
      query_1 : Struct
         product_level : DInt;
         Interface_level : DInt;
         roof_level : DInt;
         temperature : Array[1..5] of DInt;
         temperature_avg : DInt;
      END_STRUCT;
   END_VAR
BEGIN
   // MTS sensors - M-Series - Liquid-Level Sensors
   // Web: http://www.mtssensors.com/fileadmin/media/pdfs/550791.pdf

   "mb_station_block_header"(sb := #sb, mb_query := #mb_query);
   #mb_query.mb_addr := #mb_addr;

   #mb_query.mode := #mb_query.c.mode.read;
   #mb_query(data_addr := 30001,
             data_ptr := #query_1);

   "mb_station_block_footer"(sb := #sb, mb_query := #mb_query);

   #level := DINT_TO_REAL(#query_1.product_level) * 0.001;
   #temperature := DINT_TO_REAL(#query_1.temperature_avg) * 0.0001;
END_FUNCTION_BLOCK

FUNCTION_BLOCK "Novus_tht"   // FB38, SCL
{ S7_Optimized_Access := 'TRUE' }
VERSION : 0.1
   VAR_INPUT
      mb_addr : USInt;
   END_VAR
   VAR_OUTPUT
      temperature : Int;
      humidity : Int;
   END_VAR
   VAR_IN_OUT
      mb_query : "mb_query";
   END_VAR
   VAR
      sb : "mb_station_block_udt";
      serial_number : DWord;
      raw_values : Struct
         temp : Int;
         hum : Int;
      END_STRUCT;
   END_VAR
BEGIN
   // - Novus - RHT (Temperature transmitter)
   // - http://www.novusautomation.com/downloads/Arquivos/v10x_b_manual_rht_wm-dm-p10_485_lcd_%20english.pdf

   "mb_station_block_header"(sb := #sb, mb_query := #mb_query);
   #mb_query.mb_addr := #mb_addr;

   #mb_query.mode := #mb_query.c.read.holding_reg;
   #mb_query(data_addr := 7, data_ptr := #raw_values);
   #mb_query(data_addr := 0, data_ptr := #serial_number);

   "mb_station_block_footer"(sb := #sb, mb_query := #mb_query);

   #temperature := #raw_values.temp / 10;
   #humidity := #raw_values.hum / 10;
END_FUNCTION_BLOCK

FUNCTION_BLOCK "Onicon_F5100"   // FB39, SCL
{ S7_Optimized_Access := 'TRUE' }
VERSION : 0.1
   VAR_INPUT
      mb_addr : USInt;
   END_VAR
   VAR_IN_OUT
      mb_query : "mb_query";
   END_VAR
   VAR
      sb : "mb_station_block_udt";
      reset : Bool;
      query1 : Struct
         flow_total : UDInt;
      END_STRUCT;
      query2 : Struct
         flow_rate : Real;
         temperature : Real;
      END_STRUCT;
   END_VAR
BEGIN
   // Onicon - F-5100
   // http://www.onicon.com/pdfs/0669-7-F-5100-MOD-Network-Interface-Installation-Guide-09-15.pdf

   "mb_station_block_header"(sb := #sb,
                             mb_query := #mb_query);
   #mb_query.mb_addr := #mb_addr;

   #mb_query.data_addr := 312; // 313 - 1
   IF #reset THEN
       #query1.flow_total := 0;
       #mb_query(mode := #mb_query.c.write.holding_reg,
                 data_ptr := #query1.flow_total);
       IF #mb_query.stat.done THEN
           #reset := false;
       END_IF;
   ELSE
       #mb_query(mode := #mb_query.c.read.holding_reg,
                 data_ptr := #query1);
   END_IF;

   #mb_query(mode := #mb_query.c.read.holding_reg,
             data_addr := 578, // 579 - 1,
             data_ptr := #query2);

   "mb_station_block_footer"(sb := #sb,
                             mb_query := #mb_query);
END_FUNCTION_BLOCK

FUNCTION_BLOCK "Phoenix_Contact_UPS"   // FB40, SCL
{ S7_Optimized_Access := 'TRUE' }
VERSION : 0.1
   VAR_INPUT
      mb_addr : UInt;
   END_VAR
   VAR_IN_OUT
      mb_query : "mb_query";
   END_VAR
   VAR
      sb : "mb_station_block_udt";
      read1 : Struct
         remote : Word;
         BatteryMode : Word;
         ShutdownEvent : Word;
         BatteryCharging : Word;
      END_STRUCT;
      read2 : Struct
         OutputVoltage_mV : UInt;
      END_STRUCT;
      read3 : Struct
         SocStateOfCharge : UInt;   // [%]
         SocResidualBackupTimeM : UInt;   // Minute
      END_STRUCT;
      read4 : Struct
         BatteryVoltage_mV : UInt;
         BatteryTemperature : UInt;   // Kelvin
         OutputVoltage2_mV : UInt;
         SocResidualBackupTimeS : UInt;
         BatteryNomCapacityWs : UInt;
      END_STRUCT;
      read5 : Struct
         BatteryDischaCurrent : UInt;
         BatteryDetectedUnits : UInt;
         BatteryNomCapacitymAh : UInt;
         BatteryInstalledType : UInt;
      END_STRUCT;
      read6_Alarm : Struct
         x08 : Bool;
         x09_no_battery : Bool;
         x10_inconsistent_technology : Bool;
         x11_overload_cutoff : Bool;
         "x12_Low_battery_(Voltage)" : Bool;
         "x13_Low_battery_(Charge)" : Bool;
         "x14_Low_battery_(Time)" : Bool;
         x15 : Bool;
         "x00_End_of_life_(SOH)" : Bool;
         x01 : Bool;
         x02 : Bool;
         x03 : Bool;
         "x04_End_of_life_(Resitance)" : Bool;
         "x05_Endof_life_(Resitance)" : Bool;
         "x06_End_of_life_(Time)" : Bool;
         "x07_End_of_life_(Voltage)" : Bool;
      END_STRUCT;
   END_VAR
BEGIN
   // Phoenix Contact - UPS
   // QUINT UPS-IQ, TRIO-UPS
   // Web: https://media.digikey.com/pdf/Data%20Sheets/
   //      Phoenix%20Contact%20PDFs/2320461_Ds.pdf

   "mb_station_block_header"(sb := #sb, mb_query := #mb_query);
   #mb_query.mb_addr := #mb_addr;

   #mb_query.mode := #mb_query.c.read.holding_reg;
   #mb_query(data_addr := 29696, data_ptr := #read1);
   #mb_query(data_addr := 29745, data_ptr := #read2);
   #mb_query(data_addr := 29749, data_ptr := #read3);
   #mb_query(data_addr := 29792, data_ptr := #read4);
   #mb_query(data_addr := 29798, data_ptr := #read5);
   #mb_query(data_addr := 29840, data_ptr := #read6_Alarm);

   "mb_station_block_footer"(sb := #sb, mb_query := #mb_query);
END_FUNCTION_BLOCK

FUNCTION_BLOCK "Rotork_Mk_3_option_card"   // FB44, SCL
{ S7_Optimized_Access := 'TRUE' }
VERSION : 0.1
   VAR_INPUT
      mb_addr : UInt;
   END_VAR
   VAR_IN_OUT
      mb_query : "mb_query";
   END_VAR
   VAR
      sb : "mb_station_block_udt";
      read1 : Struct
         x00_actuator_moving : Bool;
         "x01_Close position limit" : Bool;
         "x02_Open position limit" : Bool;
         "x03_Valve running close" : Bool;
         "x04_Valve running open" : Bool;
         "x05_Selector in remote" : Bool;
         "x06_Selector in local stop" : Bool;
         "x07_Selector in local" : Bool;
         "x08_Thermostat tripped" : Bool;
         "x09_Monitor relay" : Bool;
         "x10_Valve obstructed" : Bool;
         "x11_Valve jammed" : Bool;
         "x12_Manual movement" : Bool;
         "x13_MIT_Interrupter timer" : Bool;
         "x14_Position control enabled" : Bool;
         "x15_Watchdog Recovery" : Bool;
         "x16_Battery low" : Bool;
         "x17_Open Interlock input active" : Bool;
         "x18_Close Interlock input active" : Bool;
         "x19_Hard wired input DI-1 (open)" : Bool;
         "x20_Hard wired input DI-2 (close)" : Bool;
         "x21_Hard wired input DI-3 (stop)" : Bool;
         "x22_Hard wired input DI-4 (ESD)" : Bool;
         x23 : Bool;
         x24 : Bool;
         x25 : Bool;
         "x26_Control contention" : Bool;
         "x27_Partial stroke test in progress" : Bool;
         "x28_Partial stroke test error" : Bool;
         "x29_General alarm" : Bool;
         x30 : Bool;
         x31 : Bool;
      END_STRUCT;
      read2 : Struct
         instantaneous_torque : Int;
         valve_position : Int;   // x10 %
         analogue_input : Int;
      END_STRUCT;
      write1 : Struct
         stop : Bool;
         close : Bool;
         open : Bool;
         emergency_shut_down : Bool;
         output_DO_1 : Bool;
         output_DO_2 : Bool;
         output_DO_3 : Bool;
         output_DO_4 : Bool;
      END_STRUCT;
      write2 : Struct
         actuator_digital_control : Bool;
         position_demand_output : Bool;
      END_STRUCT;
      actuator_tag_name : String[12];
      action_on_loss_of_comms : Int;
   END_VAR
BEGIN
   // Rotork  - Mk 3 Option Card

   // http://www.rotork.com/en/product/index/modbusliterature
   // Publication PUB091-004-00_0715

   "mb_station_block_header"(sb := #sb, mb_query := #mb_query);
   #mb_query.mb_addr := #mb_addr;

   #mb_query.mode := #mb_query.c.read.discrete_input;
   #mb_query(data_addr := 0, data_ptr := #read1);

   #mb_query.mode := #mb_query.c.read.holding_reg;
   #mb_query(data_addr := 2, data_ptr := #read2);
   #mb_query(data_addr := 26, data_ptr := #actuator_tag_name);

   #mb_query.mode := #mb_query.c.write.discrete_output;
   #mb_query(data_addr := 0, data_ptr := #write1);

   #mb_query.mode := #mb_query.c.write.holding_reg;
   // 0=No-Action, 1=Open, 3=Close, 5=Stop, 7=Position
   #mb_query(data_addr := 7, data_ptr := #action_on_loss_of_comms);
   #mb_query(data_addr := 5, data_ptr := #write2);

   "mb_station_block_footer"(sb := #sb, mb_query := #mb_query);
END_FUNCTION_BLOCK

FUNCTION_BLOCK "SensorsONE_DCT_531"   // FB52, SCL
{ S7_Optimized_Access := 'TRUE' }
VERSION : 0.1
   VAR_INPUT
      mb_addr : UInt;
   END_VAR
   VAR_IN_OUT
      mb_query : "mb_query";
   END_VAR
   VAR
      sb : "mb_station_block_udt";
      data : Struct
         serial_number : UDInt;
         date_last_calibration : UDInt;
         upper_range_pressure : Real;
         lower_range_pressure : Real;
         actual_pressure : Real;
         max_pressure : Real;
         min_pressure : Real;
         upper_range_temperature : Real;
         lower_range_temperature : Real;
         actual_temperature : Real;
         max_temperature : Real;
         min_temperature : Real;
      END_STRUCT;
   END_VAR
BEGIN
   // SensorsONE - DCT 531
   // 
   // https://www.sensorsone.com/dct-531-modbus-rtu-rs485-pressure-sensor/

   "mb_station_block_header"(sb := #sb,
                             mb_query := #mb_query);
   #mb_query.mb_addr := #mb_addr;

   #mb_query.mode := #mb_query.c.read.input_reg;
   #mb_query(data_addr := 0,
             data_ptr := #data);

   "mb_station_block_footer"(sb := #sb,
                             mb_query := #mb_query);
END_FUNCTION_BLOCK

FUNCTION_BLOCK "Sierra_thermal_mass_flow_meters"   // FB61, SCL
{ S7_Optimized_Access := 'TRUE' }
VERSION : 0.1
   VAR_INPUT
      mb_addr : UInt;
      reset_totalizer : Bool := 1;
   END_VAR
   VAR_IN_OUT
      mb_query : "mb_query";
   END_VAR
   VAR
      sb : "mb_station_block_udt";
      data : Struct
         flow : Real;
         totalizer : DInt;
      END_STRUCT;
      serial_number : String[12];
   END_VAR
   VAR_TEMP
      "int" : Int;
   END_VAR
BEGIN
   // Sierra - 600/700 Series - Thermal mass flow meters
   // Models: 620S, 620S-BT, 640S, 760S, 780S, and 780S-UHP

   // Web: https://www.ccontrols.com/support/dp/600-700-modbus-instruction-manual.pdf

   "mb_station_block_header"(sb := #sb,
                             mb_query := #mb_query);
   #mb_query.mb_addr := #mb_addr;

   #mb_query.mode := #mb_query.c.mode.read;
   #mb_query(data_addr := 40001,
             data_ptr := #data);
   #mb_query(data_addr := 40016,
             data_ptr := #serial_number);

   IF #reset_totalizer THEN
       #mb_query.mode := #mb_query.c.mode.write;
       #"int" := 1;
       #mb_query(data_addr := 40008,
                 data_ptr := #"int");
   END_IF;

   "mb_station_block_footer"(sb := #sb,
                             mb_query := #mb_query);
END_FUNCTION_BLOCK

FUNCTION_BLOCK "Smart_biene_sb_hl"   // FB62, SCL
{ S7_Optimized_Access := 'TRUE' }
VERSION : 0.1
   VAR_INPUT
      mb_addr : UInt;
   END_VAR
   VAR_IN_OUT
      mb_query : "mb_query";
   END_VAR
   VAR
      s : "mb_station_block_udt";
      data : Struct
         "Min measuring range" : Word;
         "Max measuring range" : Word;
         "Pressure Value" : Word;
         "High Pressure" : Word;
         "Low Pressure" : Word;
         stat : Word;
         model : String[12];
         serial : String[12];
         unit : Int;
      END_STRUCT;
      "a" : Struct
         x08 : Bool;
         x09 : Bool;
         x10 : Bool;
         x11 : Bool;
         x12 : Bool;
         x13 : Bool;
         x14 : Bool;
         x15 : Bool;
         x00 : Bool;
         x01 : Bool;
         x02 : Bool;
         x03 : Bool;
         x04 : Bool;
         x05 : Bool;
         x06 : Bool;
         x07 : Bool;
      END_STRUCT;
   END_VAR
BEGIN
   // Smart Biene - SB-HL - Hydrostatic Level Transmitter
   // 
   // Web: http://smartbiene.com/images/pdf/hydrostatic-level/
   //      Hydrostatic%20level-SP-HL-01-ModbusRTU.pdf

   "mb_station_block_header"(sb := #s,
                             mb_query := #mb_query);
   #mb_query.mb_addr := #mb_addr;

   #mb_query.mode := #mb_query.c.read.holding_reg;
   #mb_query(data_addr := 0,
             data_ptr := #data);

   "mb_station_block_footer"(sb := #s,
                             mb_query := #mb_query);

   (*
   Unit:
   0-mbar
   1-bar
   2-PSI
   3-KPa
   4-MPa
   5-Kg/cm2
   6-mmHg
   7-mmH2O
   8-inHg
   9-inH2O 
   *)
END_FUNCTION_BLOCK

FUNCTION_BLOCK "Socomec_diris"   // FB63, SCL
{ S7_Optimized_Access := 'TRUE' }
VERSION : 0.1
   VAR_INPUT
      mb_addr : USInt;
      old_mapping : Bool;
      zero_comm_err : Bool;
   END_VAR
   VAR_OUTPUT
      data : Struct
         voltage_L_L : Array[1..3] of Real;   // 1->L1-L2, 2->L2-L3, 3->L3-L1
         voltage_L_N : Array[1..3] of Real;
         frequency : Real;
         current : Array[1..3] of Real;
         neutral_current : Real;
         sum_active_power : Real;
         sum_reactive_power : Real;
         sum_apparent_power : Real;
         sum_power_factor : Real;   // -: leading and + : lagging
         power_active : Array[1..3] of Real;
         power_reactive : Array[1..3] of Real;
         power_apparent : Array[1..3] of Real;
         power_factor : Array[1..3] of Real;
      END_STRUCT;
   END_VAR
   VAR_IN_OUT
      mb_query : "mb_query";
   END_VAR
   VAR
      sb : "mb_station_block_udt";
      read2_temperature : DInt;
   END_VAR
   VAR_TEMP
      c : Int;
      read1 : Struct
         voltage_L_L : Array[1..3] of DInt;   // 1->L1-L2, 2->L2-L3, 3->L3-L1
         voltage_L_N : Array[1..3] of DInt;
         frequency : DInt;
         current : Array[1..3] of DInt;
         neutral_current : DInt;
         sum_active_power : DInt;
         sum_reactive_power : DInt;
         sum_apparent_power : DInt;
         sum_power_factor : DInt;   // -: leading and + : lagging
         power_active : Array[1..3] of DInt;
         power_reactive : Array[1..3] of DInt;
         power_apparent : Array[1..3] of DInt;
         power_factor : Array[1..3] of DInt;
      END_STRUCT;
   END_VAR
BEGIN
   // Socomec Diris A40/A41 - Power meter
   // https://www.socomec.com/files/live/sites/systemsite/files/SCP/
   // 6_gestion_energie/diris/diris_a40/536181B_GB_Ethernet.pdf

   // old_mapping:
   // http://www.ferrazshawmutsales.com/pdfs/cdr_27038_RS485_JBus-ModBus.pdf

   "mb_station_block_header"(sb := #sb, mb_query := #mb_query);
   #mb_query.mb_addr := #mb_addr;
   #mb_query.mode := #mb_query.c.read.holding_reg;

   #mb_query(data_addr := SEL(G := #old_mapping, IN0 := 50514, IN1 := 768),
             data_ptr := #read1);
   IF #mb_query.Done THEN
       FOR #c := 1 TO 3 DO
           #data.voltage_L_L[#c] := DINT_TO_REAL(#read1.voltage_L_L[#c]) / 100;
           #data.voltage_L_N[#c] := DINT_TO_REAL(#read1.voltage_L_N[#c]) / 100;
           #data.current[#c] := DINT_TO_REAL(#read1.current[#c]) / 1000;
           #data.power_active[#c] := DINT_TO_REAL(#read1.power_active[#c]) / 100;
           #data.power_reactive[#c] := DINT_TO_REAL(#read1.power_reactive[#c]) / 100;
           #data.power_apparent[#c] := DINT_TO_REAL(#read1.power_apparent[#c]) / 100;
           #data.power_factor[#c] := DINT_TO_REAL(#read1.power_factor[#c]) / 1000;
       END_FOR;
       #data.frequency := DINT_TO_REAL(#read1.frequency) / 100;
       #data.neutral_current := DINT_TO_REAL(#read1.neutral_current) / 100;
       #data.sum_active_power := DINT_TO_REAL(#read1.sum_active_power) / 100;
       #data.sum_reactive_power := DINT_TO_REAL(#read1.sum_reactive_power) / 100;
       #data.sum_apparent_power := DINT_TO_REAL(#read1.sum_apparent_power) / 100;
       #data.sum_power_factor := DINT_TO_REAL(#read1.sum_power_factor) / 1000;
   END_IF;

   IF NOT #old_mapping THEN
       #mb_query(data_addr := 51457, data_ptr := #read2_temperature);
   END_IF;

   "mb_station_block_footer"(sb := #sb, mb_query := #mb_query);

   IF #zero_comm_err AND #sb.out.communication_error THEN
       FOR #c := 1 TO 3 DO
           #data.voltage_L_L[#c] := 0;
           #data.voltage_L_N[#c] := 0;
           #data.current[#c] := 0;
           #data.power_active[#c] := 0;
           #data.power_reactive[#c] := 0;
           #data.power_apparent[#c] := 0;
           #data.power_factor[#c] := 0;
       END_FOR;
       #data.frequency := 0;
       #data.neutral_current := 0;
       #data.sum_active_power := 0;
       #data.sum_reactive_power := 0;
       #data.sum_apparent_power := 0;
       #data.sum_power_factor := 0;

       #read2_temperature := 0;
   END_IF;
END_FUNCTION_BLOCK

FUNCTION_BLOCK "Sparling_Instruments_Tiger_Mag"   // FB64, SCL
{ S7_Optimized_Access := 'TRUE' }
VERSION : 0.1
   VAR_INPUT
      mb_addr : USInt;
   END_VAR
   VAR_IN_OUT
      mb_query : "mb_query";
   END_VAR
   VAR
      sb : "mb_station_block_udt";
      read1 : Struct
         flow : Real;   // 0.01 [Hz]
         total_fwd : UDInt;   // 0.1 [A]
         total_rev : UDInt;
         unit_flow : String[4];
         unit_total : String[4];
         total_registration : Real;
      END_STRUCT;
      serial_number : UDInt;
   END_VAR
BEGIN
   // Sparling Instruments - Tiger Mag 
   // FM656, FM657, FM626, FM627, FM626 Sanitary
   // http://www.sparlinginstruments.com/documents/IDS-TMEP-160323.PDF
   // Revision 160323

   "mb_station_block_header"(sb := #sb,
                             mb_query := #mb_query);
   #mb_query.mb_addr := #mb_addr;

   #mb_query.mode := #mb_query.c.mode.read;
   #mb_query(data_addr := 30001,
             data_ptr := #read1);
   #mb_query(data_addr := 31003,
             data_ptr := #serial_number);

   "mb_station_block_footer"(sb := #sb,
                             mb_query := #mb_query);

   (*
   Terminal RS-485 Bus:
   1-RX  -> A+
   2-TX  -> B-
   3-GND -> GND
   4-DTR -> N/A Not used

   Default comm. param:
   19200 bps, even parity. 
    Slave ID: 1.
   *)
END_FUNCTION_BLOCK

FUNCTION_BLOCK "Syxthsense_TEHR_M"   // FB70, SCL
TITLE = Syxthsense - TEHR-M - Temperature transmitter
{ S7_Optimized_Access := 'TRUE' }
AUTHOR : OlaBjornli
VERSION : 0.1
   VAR_INPUT
      mb_addr : USInt := 1;
   END_VAR
   VAR_OUTPUT
      temperature : Real;   // [Â°C]
      analogue_output : Real;   // [Â°F]
      potentiometer_position : Real;   // [%]
   END_VAR
   VAR_IN_OUT
      mb_query : "mb_query";
   END_VAR
   VAR
      sb : "mb_station_block_udt";
      read1 : Struct
         temperature : Int;   // [Â°C]
         analogue_output : Int;   // [Â°F]
         potentiometer_position : Int;   // [%]
      END_STRUCT;
   END_VAR
BEGIN
   // http://www.syxthsense.com/product/product_pdf/SN1.174-TEHR-M.pdf

   "mb_station_block_header"(sb := #sb, mb_query := #mb_query);

   #mb_query(mb_addr := #mb_addr,
             mode := #mb_query.c.mode.read,
             data_addr := 30001,
             data_ptr := #read1);
   #temperature := INT_TO_REAL(#read1.temperature) / 10;
   #analogue_output := INT_TO_REAL(#read1.analogue_output) / 10;
   #potentiometer_position := INT_TO_REAL(#read1.potentiometer_position) / 10;

   "mb_station_block_footer"(sb := #sb, mb_query := #mb_query);
END_FUNCTION_BLOCK

FUNCTION_BLOCK "Vacon_OPTC2_C8"   // FB72, SCL
{ S7_Optimized_Access := 'TRUE' }
VERSION : 0.1
   VAR_INPUT
      mb_addr : UInt;
      ref : Real;
   END_VAR
   VAR_OUTPUT
      actual_speed : Real;
      Output_Frequency : Real;   // hz
      Motor_Speed : Real;   // rpm
      Motor_Current : Real;   // A
      Motor_Torque : Real;   // %
      Motor_Power : Real;   // %
      Motor_Voltage : Real;   // V
      DC_link_voltage : Real;   // V
   END_VAR
   VAR_IN_OUT
      mb_query : "mb_query";
   END_VAR
   VAR
      sb : "mb_station_block_udt";
      write : Struct
         ctw : Struct
            byte0 : Bool;
            x00_run : Bool;
            x01_reverse : Bool;
            x02_reset : Bool;
            x03 : Bool;
            x04 : Bool;
            x05 : Bool;
            x06 : Bool;
            x07 : Bool;
         END_STRUCT;
         "General Control Word" : Word;
         speed_reference : Int;
      END_STRUCT;
      read : Struct
         status : Struct
            x08_TC_Speed_Limit_Not_Active : Bool;
            x09_Detected_Encoder_Direction_Counterclockwise : Bool;
            x10_UV_Fast_Stop_Not_Active : Bool;
            x11 : Bool;
            x12 : Bool;
            x13 : Bool;
            x14 : Bool;
            x15 : Bool;
            x00_ready : Bool;
            x01_RUN : Bool;
            x02_reverse : Bool;
            x03_Faulted : Bool;
            x04_Warning : Bool;
            x05_Ref_Frequency_reached : Bool;
            x06_Motor_is_running_at_zero_speed : Bool;
            x07_Flux_Ready : Bool;
         END_STRUCT;
         general_status : Struct
            x08 : Bool;
            x09 : Bool;
            x10 : Bool;
            x11 : Bool;
            x12 : Bool;
            x13_Fieldbus_control : Bool;
            "x14_Panel control" : Bool;
            x15_IO_control : Bool;
            x00 : Bool;
            x01 : Bool;
            x02 : Bool;
            x03 : Bool;
            x04 : Bool;
            x05 : Bool;
            x06 : Bool;
            x07 : Bool;
         END_STRUCT;
         actual_speed : Int;
         Output_Frequency : Int;   // 0.01 Hz
         Motor_Speed : Int;   // 1 rpm
         Motor_Current : Int;   // 0.1 A
         Motor_Torque : Int;   // 0.1 %
         Motor_Power : Int;   // 0.1 %
         Motor_Voltage : Int;   // 0.1 V
         DC_link_voltage : Int;   // 1 V
         Active_Fault_Code : Int;
      END_STRUCT;
   END_VAR
BEGIN
   // Vacon NX - OPTC2/C8 - AC drives
   // Modbus/N2 option board
   // Document code: DPD00899A , Date 19.01.2012
   // Web: http://www.vacon.com/ImageVaultFiles/id_3118/cf_2/
   //      Vacon-NX-OPTC2-C8-Modbus-N2-Board-User-Manual-DPD0.
   //      PDF?635223804391930000

   "mb_station_block_header"(sb := #sb, mb_query := #mb_query);
   #mb_query.mb_addr := #mb_addr;

   #mb_query.mode := #mb_query.c.read.holding_reg;

   #mb_query(data_addr := 42101, data_ptr := #read);
   #actual_speed := INT_TO_REAL(#read.actual_speed);
   #Output_Frequency := INT_TO_REAL(#read.Output_Frequency) * 0.01;
   #Motor_Speed := INT_TO_REAL(#read.Motor_Speed);
   #Motor_Current := INT_TO_REAL(#read.Motor_Current) * 0.1;
   #Motor_Torque := INT_TO_REAL(#read.Motor_Torque) * 0.1;
   #Motor_Power := INT_TO_REAL(#read.Motor_Power) * 0.1;
   #Motor_Voltage := INT_TO_REAL(#read.Motor_Voltage) * 0.1;
   #DC_link_voltage := INT_TO_REAL(#read.DC_link_voltage);

   // -------------------------------------------------------
   #mb_query.mode := #mb_query.c.write.holding_reg;

   #write.ctw.x00_run := #ref <> 0;
   #mb_query(data_addr := 42001, data_ptr := #write.ctw);
   #write.speed_reference := REAL_TO_INT(#ref * 100);
   #mb_query(data_addr := 42003, data_ptr := #write.speed_reference);

   "mb_station_block_footer"(sb := #sb, mb_query := #mb_query);
END_FUNCTION_BLOCK

FUNCTION_BLOCK "vega_vegabar_81"   // FB73, SCL
{ S7_Optimized_Access := 'TRUE' }
VERSION : 0.1
   VAR_INPUT
      mb_addr : UInt;
   END_VAR
   VAR_IN_OUT
      mb_query : "mb_query";
   END_VAR
   VAR
      sb : "mb_station_block_udt";
      read1 : Struct
         status : Struct
            x08 : Bool;
            x09 : Bool;
            x10 : Bool;
            x11 : Bool;
            x12 : Bool;
            x13 : Bool;
            x14 : Bool;
            x15 : Bool;
            x00_invalid_measurement_1 : Bool;
            x01_invalid_measurement_2 : Bool;
            x02_invalid_measurement_3 : Bool;
            x03_invalid_measurement_4 : Bool;
            x04 : Bool;
            x05 : Bool;
            x06 : Bool;
            x07 : Bool;
         END_STRUCT;
         z : Word;
         data : Array[1..4] of Real;
      END_STRUCT;
   END_VAR
BEGIN
   // Vega - VEGABAR 81

   "mb_station_block_header"(sb := #sb, mb_query := #mb_query);
   #mb_query.mb_addr := #mb_addr;

   #mb_query(mode := #mb_query.c.read.holding_reg,
             data_addr := 2000,
             data_ptr := #read1);

   "mb_station_block_footer"(sb := #sb, mb_query := #mb_query);

   (*
   Unit Code Measurement Unit:
   32 Degree Celsius
   33 Degree Fahrenheit
   40 US Gallon
   41 Liters
   42 Imperial Gallons
   43 Cubic Meters
   44 Feet
   45 Meters
   46 Barrels
   47 Inches
   48 Centimeters
   49 Millimeters
   111 Cubic Yards
   112 Cubic Feet
   113 Cubic Inches
   *)
END_FUNCTION_BLOCK

FUNCTION_BLOCK "Weg_CFW100"   // FB74, SCL
{ S7_Optimized_Access := 'TRUE' }
VERSION : 0.1
   VAR_INPUT
      mb_addr : UInt;
   END_VAR
   VAR_IN_OUT
      mb_query : "mb_query";
   END_VAR
   VAR
      sb : "mb_station_block_udt";
      r1 : Struct
         Output_Speed : UInt;   // 2
         Motor_Current : UInt;
         DC_Link_Voltage : UInt;
         Output_Frequency : UInt;
         Inverter_Status : UInt;
         Output_Voltage : UInt;
         Motor_Torque : UInt;
         Active_Current : UInt;
         digital_input : UInt;
      END_STRUCT;
      r2_staus : Struct
         x08_running : Bool;
         x09_ready : Bool;
         x10_forward : Bool;
         x11_jog_active : Bool;
         x12_remote_mode : Bool;
         x13_undervoltage : Bool;
         x14_ : Bool;
         x15_fault : Bool;
         x00 : Bool;
         x01 : Bool;
         x02 : Bool;
         x03 : Bool;
         x04 : Bool;
         x05_2nd_Ramp : Bool;   // 0: 1st Acceleration and deceleration ramp by P100 and P101.
         x06_configuration_state : Bool;
         x07_alarm : Bool;
         "a" : Struct
            x08 : Bool;
            x09 : Bool;
            x10 : Bool;
            x11 : Bool;
            x12 : Bool;
            x13 : Bool;
            x14 : Bool;
            x15 : Bool;
            x00 : Bool;
            x01 : Bool;
            x02 : Bool;
            x03 : Bool;
            x04 : Bool;
            x05 : Bool;
            x06 : Bool;
            x07 : Bool;
         END_STRUCT;
      END_STRUCT;
      _ : Bool;
      w1 : Struct
         Minimum_Frequency : UInt;
         Maximum_Frequency : UInt := 50;
         Maximum_Output_Current : UInt := 100;
      END_STRUCT;
      w2 : Struct
         "Acceleration Time" : UInt := 5;
         "Deceleration Time" : UInt := 10;
      END_STRUCT;
      w3_sel_rem : UInt := 1;   // 1 = Always Remote
      w4_Ref_sel : UInt := 9;   // 9=serial
      w5 : Struct
         controll_word : Struct
            x08 : Bool;
            x09 : Bool;
            x10 : Bool;
            x11 : Bool;
            x12 : Bool;
            x13 : Bool;
            x14 : Bool;
            x15 : Bool;
            x00_no_ramp_stop : Bool := TRUE;
            x01_start : Bool := TRUE;
            x02_Forward : Bool;
            x03_jog : Bool;
            x04_Remote : Bool := TRUE;
            "x05_2nd Ramp" : Bool;
            x06 : Bool;
            x07_Fault_Reset : Bool;
            "a" : Struct
               x08 : Bool;
               x09 : Bool;
               x10 : Bool;
               x11 : Bool;
               x12 : Bool;
               x13 : Bool;
               x14 : Bool;
               x15 : Bool;
               x00 : Bool;
               x01 : Bool;
               x02 : Bool;
               x03 : Bool;
               x04 : Bool;
               x05 : Bool;
               x06 : Bool;
               x07 : Bool;
            END_STRUCT;
         END_STRUCT;
         speed_ref : Int;
      END_STRUCT;
      w6_stop_mode : Int;
      w7_no_comm_action : Int := 1;   // 1 = Ramp Stop
      c : Int := 1;
      setup_finished : Bool;
   END_VAR
BEGIN
   // Weg - CFW100
   // 
   // Web: http://www.clrwtr.com/PDF/WEG/WEG-CFW100-Programming.pdf

   "mb_station_block_header"(sb := #sb,
                             mb_query := #mb_query);
   #mb_query.mb_addr := #mb_addr;

   #mb_query.mode := #mb_query.c.read.holding_reg;
   #mb_query(data_addr := 2,
             data_ptr := #r1);
   #mb_query(data_addr := 680,
             data_ptr := #r2_staus);

   #mb_query.mode := #mb_query.c.write.holding_reg;
   #mb_query(data_addr := 682,
             data_ptr := #w5);
   CASE #c OF
       1:
           #mb_query(data_addr := 133,
                     data_ptr := #w1);
       2:
           #mb_query(data_addr := 101,
                     data_ptr := #w2);
       3:
           #mb_query(data_addr := 220,
                     data_ptr := #w3_sel_rem);
       4:
           #mb_query(data_addr := 222,
                     data_ptr := #w4_Ref_sel);
       5:
           #mb_query(data_addr := 229,
                     data_ptr := #w6_stop_mode);
       6:
           #mb_query(data_addr := 313,
                     data_ptr := #w7_no_comm_action);
       ELSE:
           #c := 0;
   END_CASE;
   #c += BOOL_TO_INT(#mb_query.Done);

   "mb_station_block_footer"(sb := #sb,
                             mb_query := #mb_query);
   IF #sb.out.communication_error THEN
       #setup_finished := false;
   END_IF;

   (*
   P229 Stop mode:
   0 The inverter will apply the stop ramp programmed in P101 or P103.
   1 The motor will run free until it stops

   P006 Inverter Status:
   0 = Ready
   1 = Run
   2 = Undervoltage
   3 = Fault
   4 = Not Used
   5 = Configuration

   *)
END_FUNCTION_BLOCK

FUNCTION_BLOCK "Wika_GDT20_GDHT20"   // FB75, SCL
{ S7_Optimized_Access := 'TRUE' }
VERSION : 0.1
   VAR_INPUT
      mb_addr : UInt;
   END_VAR
   VAR_IN_OUT
      mb_query : "mb_query";
   END_VAR
   VAR
      sb : "mb_station_block_udt";
      data : Struct
         pressure_bar : Real;
         pressure_MPa : Real;
         pressure_Pa : Real;
         pressure_kPa : Real;
         pressure_psi : Real;
         pressure_N_cmÂ² : Real;
         Temperature_C : Real;
         Temperature_K : Real;
         Temperature_F : Real;
         gas_density_g_l : Real;
         gas_density_kg_m3 : Real;
         "Pressure_standardised_to 20_C" : Real;
         Humidity_Atmosphere_frost_point : Real;
         Humidity_Atmosphere_dew_point : Real;
         Humidity_Tank_pressure_frost_point : Real;
         Humidity_Tank_pressure_dew_point_1 : Real;
      END_STRUCT;
      tag : String[16];
      alarm : Struct
         x08_Failure_humidity_sensor : Bool;   // (only model GDHT-20)
         x09_Communication_error_humidity_sensor : Bool;   // (only model GDHT-20)
         x10_Re_occurring_Modbus_communication_error : Bool;   // Re-occurring ModbusÂ® communication error
         x11 : Bool;
         x12 : Bool;
         x13 : Bool;
         x14 : Bool;
         x15 : Bool;
         x00_Pressure_below_lower_limit : Bool;   // Pressure signal below the lower limit value (< 0 bar)
         x01_Pressure_above_upper_limit : Bool;
         x02_Pressure_sensor_failure : Bool;
         x03_Temperature_below_lower_limit : Bool;   // Temperature signal below the lower limit value (< -40 Â°C)
         x04_Temperature_above_upper_limit : Bool;
         x05_Communication_error_pressure_temperature_sensor : Bool;
         x06_Pressure_density_below_lower_limit : Bool;   // Pressure density below the lower limit value (liquefaction of SF6 gas)
         x07_Gas_density_above_upper_limit : Bool;   // Gas density above the upper limit value (> 80 g/l)
      END_STRUCT;
      reset_alarm : Bool;
   END_VAR
   VAR_TEMP
      "int" : Int;
   END_VAR
BEGIN
   // Wika - GDT-20, GDHT-20 (GDT-20, GDHT-20)
   // Pressure / temperature / Gas density / Humidity 
   // 
   // http://en-co.wika.de/upload/OI_GDT_GDHT_20_en_de_67032.pdf

   "mb_station_block_header"(sb := #sb,
                             mb_query := #mb_query);
   #mb_query.mb_addr := #mb_addr;

   #mb_query.mode := #mb_query.c.read.holding_reg;
   #mb_query(data_addr := 0,
             data_ptr := #data);
   #mb_query(data_addr := 113,
             data_ptr := #tag);
   #mb_query(data_addr := 200,
             data_ptr := #alarm);

   IF #reset_alarm THEN
       #"int" := 1;
       #mb_query(mode := #mb_query.c.write.holding_reg,
                 data_addr := 201,
                 data_ptr := #"int");
       IF #mb_query.Done THEN
           #reset_alarm := false;
       END_IF;
   END_IF;

   "mb_station_block_footer"(sb := #sb,
                             mb_query := #mb_query);


   (*
   Circular connector M12 x 1 (5-pin):
   1 C Reference potential RS-485 common
   2 UB Voltage supply (DC 17 ... 30 V)
   3 GND Ground
   4 A Signal RS-485
   5 B Signal RS-485
   *)
END_FUNCTION_BLOCK

FUNCTION_BLOCK "Yaskawa_e7_drive"   // FB76, SCL
{ S7_Optimized_Access := 'TRUE' }
VERSION : 0.1
   VAR_INPUT
      mb_addr : UInt;
   END_VAR
   VAR_IN_OUT
      mb_query : "mb_query";
   END_VAR
   VAR
      sb : "mb_station_block_udt";
      read1 : Struct
         stat : Struct
            x08 : Bool;
            x09 : Bool;
            x10 : Bool;
            x11 : Bool;
            x12 : Bool;
            x13 : Bool;
            x14 : Bool;
            x15 : Bool;
            x00_run : Bool;
            x01 : Bool;
            x02 : Bool;
            x03_reset_signal : Bool;
            x04_speed_agree : Bool;
            x05_inverter_ready : Bool;
            x06_minor_fault : Bool;
            x07_major_fault : Bool;
            "a" : Struct
               x08 : Bool;
               x09 : Bool;
               x10 : Bool;
               x11 : Bool;
               x12 : Bool;
               x13 : Bool;
               x14 : Bool;
               x15 : Bool;
               x00 : Bool;
               x01 : Bool;
               x02 : Bool;
               x03 : Bool;
               x04 : Bool;
               x05 : Bool;
               x06 : Bool;
               x07 : Bool;
            END_STRUCT;
         END_STRUCT;
      END_STRUCT;
      read2 : Struct
         fault_contents_1 : Struct
            x08_inverter_overheat : Bool;
            x09_inverter_overheat_warning : Bool;
            x10_motor_overload : Bool;
            x11_inverter_overload : Bool;
            x12_overtorque_1 : Bool;
            x13_overtorque_2 : Bool;
            x14_braking_resistor_fault : Bool;
            x15_braking_resistor_overheat : Bool;
            x00_fuse : Bool;
            x01_main_circuit_undervoltage : Bool;
            x02_control_circuit_undervoltage : Bool;
            x03_mc_error : Bool;
            x04 : Bool;
            x05_ground_fault : Bool;
            x06_over_current : Bool;
            x07_overvoltage : Bool;
            "a" : Struct
               x08 : Bool;
               x09 : Bool;
               x10 : Bool;
               x11 : Bool;
               x12 : Bool;
               x13 : Bool;
               x14 : Bool;
               x15 : Bool;
               x00 : Bool;
               x01 : Bool;
               x02 : Bool;
               x03 : Bool;
               x04 : Bool;
               x05 : Bool;
               x06 : Bool;
               x07 : Bool;
            END_STRUCT;
         END_STRUCT;
      END_STRUCT;
      read3_data : Struct
         "Output Frequency" : Word;   // 0.01Hz
         "Output Current" : Word;   // 0.1A
         "Output Voltage" : Word;   // 0.1Vac
         "DC Bus Voltage" : Word;   // Vdc
         "Output Power" : Word;   // 0.1kW
      END_STRUCT;
      _ : Bool;
      write1 : Struct
         cmd : Struct
            x08 : Bool;
            x09 : Bool;
            x10 : Bool;
            x11 : Bool;
            x12 : Bool;
            x13 : Bool;
            x14 : Bool;
            x15 : Bool;
            x00_run : Bool := TRUE;
            x01_reverse : Bool;
            x02_external_fault : Bool;
            x03_fault_reset : Bool;
            x04_ComNet : Bool := TRUE;
            x05_ComCtrl : Bool := TRUE;
            x06 : Bool;
            x07 : Bool;
         END_STRUCT;
         freq_ref : Int;
      END_STRUCT;
      write2_max_frequency : UInt := 50;   // 0.1 Hz
      write3 : Struct
         ref_source : Int := 2;   // 0=Operator, 1=Terminals, 2=Serial Com, 3=Option PCB
         run_source : Int := 2;   // 0=Operator, 1=Terminals, 2=Serial Com, 3=Option PCB
         stopp_method : Int := 0;   // 0=Ramp to Stop, 1=Coast to Stop, 2=DCInj to Stop, 3=Coast w/Timer (C1-09)
      END_STRUCT;
   END_VAR
BEGIN
   // Yaskawa - E7 Drive
   // Models: CIMR-E7U* 
   // Web: https://www.ccontrols.com/support/dp/TME711.pdf

   "mb_station_block_header"(sb := #sb,
                             mb_query := #mb_query);
   #mb_query.mb_addr := #mb_addr;

   #mb_query.mode := #mb_query.c.read.holding_reg;
   #mb_query(data_addr := 16#10,
             data_ptr := #read1);
   #mb_query(data_addr := 16#14,
             data_ptr := #read2);
   #mb_query(data_addr := 16#41,
             data_ptr := #read3_data);

   #mb_query.mode := #mb_query.c.write.holding_reg;
   #mb_query(data_addr := 16#303,
             data_ptr := #write2_max_frequency);
   #mb_query(data_addr := 16#180,
             data_ptr := #write3);
   #mb_query(data_addr := 16#1,
             data_ptr := #write1);

   "mb_station_block_footer"(sb := #sb,
                             mb_query := #mb_query);
END_FUNCTION_BLOCK

FUNCTION_BLOCK "Yokogawa_multivariable_transmitter"   // FB77, SCL
{ S7_Optimized_Access := 'TRUE' }
VERSION : 0.1
   VAR_INPUT
      mb_addr : UInt;
   END_VAR
   VAR_IN_OUT
      mb_query : "mb_query";
   END_VAR
   VAR
      sb : "mb_station_block_udt";
      data : Struct
         pres : Real;
         sp : Real;
         et : Real;
      END_STRUCT;
   END_VAR
BEGIN
   // Yokogawa - EJX910A and EJX930A - Multivariable Transmitter
   // web: https://web-material3.yokogawa.com/IM01C25R05-01EN_001.pdf?_ga=
   //      2.43421607.346053457.1505559574-1218156352.1505559574

   "mb_station_block_header"(sb := #sb, mb_query := #mb_query);
   #mb_query.mb_addr := #mb_addr;

   #mb_query(mode := #mb_query.c.read.input_reg,
             data_addr := 401,
             data_ptr := #data);

   "mb_station_block_footer"(sb := #sb, mb_query := #mb_query);
END_FUNCTION_BLOCK

FUNCTION_BLOCK "Accuenergy_Accuvim_L_Series_Power_meter"   // FB81, SCL
{ S7_Optimized_Access := 'TRUE' }
VERSION : 0.1
   VAR_INPUT
      mb_addr : USInt;
   END_VAR
   VAR_IN_OUT
      mb_query : "mb_query";
   END_VAR
   VAR
      sb : "mb_station_block_udt";
      read1 : Struct
         Frequency : Real;
         "Phase voltage" : Array[1..3] of Real;
         "Line voltage" : Array[1..3] of Real;
         Phase_current : Array[1..3] of Real;
         Neutral_current : Real;
         "Phase power" : Array[1..3] of Real;
         "System power Psum" : Real;
         "Phase reactive power" : Array[1..3] of Real;
         "System reactive power" : Real;
         "System apparent Ssum" : Real;
         Phase_power_factor : Array[1..3] of Real;
         "System power PFsum" : Real;
         "Voltage unbalance factor" : Real;
         "Current unbalance factor" : Real;
         _ : DWord;
         "Phase apparent power S" : Array[1..3] of Real;
         __ : DWord;
         "Apparent power demand" : Real;
         "Power demand P_Dmd" : Real;
         "Reactive power demand" : Real;
         "Phase current demand" : Array[1..3] of Real;
      END_STRUCT;
      read2_run_time : Struct
         Meter : UDInt;
         Load : UDInt;
      END_STRUCT;
      read3 : Struct
         Import_energy_Ep_imp : UDInt;
         Export_energy_Ep_exp : UDInt;
         Import_reactive_energy_Eq_imp : UDInt;
         Export_reactive_energy_Eq_exp : UDInt;
         Apparent_energy_Es : UDInt;
         Phase_energy : Array[1..3] of Struct
            "import Ep_imp" : UDInt;
            "export Ep_exp" : UDInt;
         END_STRUCT;
      END_STRUCT;
   END_VAR
BEGIN
   // Accuenergy - Accuvim-L Series Power meter
   // 
   // - https://www.accuenergy.com/files/acuvim-l/
   //   Acuvim-L-Panel-Submeter-Power-Energy-Meter-User-%20Manual(1030E2201).pdf

   "mb_station_block_header"(sb := #sb,
                             mb_query := #mb_query);
   #mb_query.mb_addr := #mb_addr;

   #mb_query.mode := #mb_query.c.read.holding_reg;
   #mb_query(data_addr := 16#600,
             data_ptr := #read1);
   #mb_query(data_addr := 16#180,
             data_ptr := #read2_run_time);
   #mb_query(data_addr := 16#156,
             data_ptr := #read3);

   "mb_station_block_footer"(sb := #sb,
                             mb_query := #mb_query);
END_FUNCTION_BLOCK

FUNCTION_BLOCK "DAE_Instrument_PM210"   // FB82, SCL
{ S7_Optimized_Access := 'TRUE' }
VERSION : 0.1
   VAR_INPUT
      mb_addr : USInt;
   END_VAR
   VAR_IN_OUT
      mb_query : "mb_query";
   END_VAR
   VAR
      sb : "mb_station_block_udt";
   END_VAR
   VAR RETAIN
      conf : Struct
         write : Bool;
         PT_ratio : Real;
         CT_ratio : Real;
      END_STRUCT;
   END_VAR
   VAR
      data1 : Struct
         voltage_Lx_N : Array[1..3] of Real;
         voltage_L_L : Array[1..3] of Real;
         current : Array[1..3] of Real;
         total_active_power : Real;
         total_reactive_power : Real;
         total_apparent_power : Real;
         frequency : Real;
         power_factor : Real;
         total_active_energy : Real;
         total_reactive_energy : Real;
         "15_minute_block_demand" : Real;
         "1_minute_block_demand" : Real;
         generator_total_active_energy : Real;
         generator_total_reactive_energy : Real;
      END_STRUCT;
      data2 : Struct
         energy_active : Struct   // VA
            phase : Array[1..3] of Real;
            total : Real;
         END_STRUCT;
         energy_reactive : Struct
            phase : Array[1..3] of Real;
            total : Real;
         END_STRUCT;
         power_active : Struct
            phase : Array[1..3] of Real;
            total : Real;
         END_STRUCT;
         power_reactive : Struct
            phase : Array[1..3] of Real;
            total : Real;
         END_STRUCT;
         power_apparent : Struct
            phase : Array[1..3] of Real;
            total : Real;
         END_STRUCT;
         power_factor : Struct
            phase : Array[1..3] of Real;
            total : Real;
         END_STRUCT;
      END_STRUCT;
      read3_temperature : Int;
      read4_io : Struct
         digital_output : Word;
         digital_input : Word;
      END_STRUCT;
      data5_generator_energy : Struct
         active : Struct
            phase : Array[1..3] of Real;
            total : Real;
         END_STRUCT;
         reactive : Struct
            phase : Array[1..3] of Real;
            total : Real;
         END_STRUCT;
      END_STRUCT;
   END_VAR
   VAR_TEMP
      read1 : Struct
         voltage_Lx_N : Array[1..3] of UDInt;   // volt
         voltage_L_L : Array[1..3] of UDInt;   // volt 1:L1-L2, 2:L2-L3, 3:L3-L1
         current : Array[1..3] of UDInt;   // mA
         total_active_power : UDInt;
         total_reactive_power : UDInt;
         total_apparent_power : UDInt;
         frequency : UDInt;
         power_factor : DInt;
         total_active_energy : UDInt;
         total_reactive_energy : UDInt;
         "15_minute_block_demand" : UDInt;
         "1_minute_block_demand" : UDInt;
         generator_total_active_energy : UDInt;
         generator_total_reactive_energy : UDInt;
      END_STRUCT;
      read2 : Struct
         energy_active : Struct   // VA
            phase : Array[1..3] of UDInt;
            total : UDInt;
         END_STRUCT;
         energy_reactive : Struct
            phase : Array[1..3] of UDInt;
            total : UDInt;
         END_STRUCT;
         power_active : Struct
            phase : Array[1..3] of UDInt;
            total : UDInt;
         END_STRUCT;
         power_reactive : Struct
            phase : Array[1..3] of UDInt;
            total : UDInt;
         END_STRUCT;
         power_apparent : Struct
            phase : Array[1..3] of UDInt;
            total : UDInt;
         END_STRUCT;
         power_factor : Struct
            phase : Array[1..3] of Int;
            total : Int;
         END_STRUCT;
      END_STRUCT;
      read5_generator_energy : Struct
         active : Struct
            phase : Array[1..3] of UDInt;
            total : UDInt;
         END_STRUCT;
         reactive : Struct
            phase : Array[1..3] of UDInt;
            total : UDInt;
         END_STRUCT;
      END_STRUCT;
      write1 : Struct
         PT_ratio : UInt;
         CT_ratio : UInt;
      END_STRUCT;
      c : Int;
   END_VAR
BEGIN
   // DAE Instrument Corp. - PM210 
   // Multi-Function Panel Meter
   //
   // Default: 9600-8-N-1
   // 
   // http://www.daeinstrument.com/downloads/PM210%20Modbus%20Reference-2.6.1e.pdf

   "mb_station_block_header"(sb := #sb, mb_query := #mb_query);
   #mb_query.mb_addr := #mb_addr;
   #mb_query.mode := #mb_query.c.read.holding_reg;

   #mb_query(data_addr := 20, data_ptr := #read1);
   IF #mb_query.Done THEN
       FOR #c := 1 TO 3 DO
           #data1.voltage_Lx_N[#c] := UDINT_TO_REAL(ROR(IN := #read1.voltage_Lx_N[#c], N := 16)) * 0.1;
           #data1.voltage_L_L[#c] := UDINT_TO_REAL(ROR(IN := #read1.voltage_L_L[#c], N := 16)) * 0.1;
           #data1.current[#c] := UDINT_TO_REAL(ROR(IN := #read1.current[#c], N := 16)) * 0.001;
       END_FOR;
       #data1.total_active_power := UDINT_TO_REAL(ROR(IN := #read1.total_active_power, N := 16));
       #data1.total_reactive_power := UDINT_TO_REAL(ROR(IN := #read1.total_reactive_power, N := 16));
       #data1.total_apparent_power := UDINT_TO_REAL(ROR(IN := #read1.total_apparent_power, N := 16));
       #data1.frequency := UDINT_TO_REAL(ROR(IN := #read1.frequency, N := 16)) * 0.1;
       #data1.power_factor := DINT_TO_REAL(ROR(IN := #read1.power_factor, N := 16)) * 0.001;
       #data1.total_active_energy := UDINT_TO_REAL(ROR(IN := #read1.total_active_energy, N := 16)) * 0.01;
       #data1.total_reactive_energy := UDINT_TO_REAL(ROR(IN := #read1.total_reactive_energy, N := 16)) * 0.01;
       #data1."15_minute_block_demand" := UDINT_TO_REAL(ROR(IN := #read1."15_minute_block_demand", N := 16)) * 0.1;
       #data1."1_minute_block_demand" := UDINT_TO_REAL(ROR(IN := #read1."1_minute_block_demand", N := 16)) * 0.1;
       #data1.generator_total_active_energy := UDINT_TO_REAL(ROR(IN := #read1.generator_total_active_energy, N := 16)) * 0.01;
       #data1.generator_total_reactive_energy := UDINT_TO_REAL(#read1.generator_total_reactive_energy) * 0.01;
   END_IF;

   #mb_query(data_addr := 80, data_ptr := #read2);
   IF #mb_query.Done THEN
       FOR #c := 1 TO 3 DO
           #data2.energy_active.phase[#c] := UDINT_TO_REAL(ROR(IN := #read2.energy_active.phase[#c], N := 16)) * 0.01;
           #data2.energy_reactive.phase[#c] := UDINT_TO_REAL(ROR(IN := #read2.energy_reactive.phase[#c], N := 16)) * 0.01;
           #data2.power_active.phase[#c] := UDINT_TO_REAL(ROR(IN := #read2.power_active.phase[#c], N := 16));
           #data2.power_reactive.phase[#c] := UDINT_TO_REAL(ROR(IN := #read2.power_reactive.phase[#c], N := 16));
           #data2.power_apparent.phase[#c] := UDINT_TO_REAL(ROR(IN := #read2.power_apparent.phase[#c], N := 16));
           #data2.power_factor.phase[#c] := INT_TO_REAL(#read2.power_factor.phase[#c]) * 0.001;
       END_FOR;
       #data2.energy_active.total := UDINT_TO_REAL(ROR(IN := #read2.energy_active.total, N := 16)) * 0.01;
       #data2.energy_reactive.total := UDINT_TO_REAL(ROR(IN := #read2.energy_reactive.total, N := 16)) * 0.01;
       #data2.power_active.total := UDINT_TO_REAL(ROR(IN := #read2.power_active.total, N := 16));
       #data2.power_reactive.total := UDINT_TO_REAL(ROR(IN := #read2.power_reactive.total, N := 16));
       #data2.power_apparent.total := UDINT_TO_REAL(ROR(IN := #read2.power_apparent.total, N := 16));
       #data2.power_factor.total := INT_TO_REAL(#read2.power_factor.total) * 0.001;
   END_IF;

   #mb_query(data_addr := 139, data_ptr := #read3_temperature);
   #mb_query(data_addr := 142, data_ptr := #read4_io);
   #mb_query(data_addr := 144, data_ptr := #read5_generator_energy);
   IF #mb_query.Done THEN
       FOR #c := 1 TO 3 DO
           #data5_generator_energy.active.phase[#c] := UDINT_TO_REAL(ROR(IN := #read5_generator_energy.active.phase[#c], N := 16)) * 0.01;
           #data5_generator_energy.reactive.phase[#c] := UDINT_TO_REAL(ROR(IN := #read5_generator_energy.reactive.phase[#c], N := 16)) * 0.01;
       END_FOR;
       #data5_generator_energy.active.total := UDINT_TO_REAL(ROR(IN := #read5_generator_energy.active.total, N := 16)) * 0.01;
       #data5_generator_energy.reactive.total := UDINT_TO_REAL(ROR(IN := #read5_generator_energy.reactive.total, N := 16)) * 0.01;
   END_IF;

   IF #conf.write THEN
       #write1.PT_ratio := REAL_TO_UINT(#conf.PT_ratio * 100);
       #write1.CT_ratio := REAL_TO_UINT(#conf.CT_ratio);
       #mb_query(mode := #mb_query.c.write.holding_reg,
                 data_addr := 133,
                 data_ptr := #write1);
       #conf.write := #conf.write AND NOT #mb_query.Done;
   END_IF;

   "mb_station_block_footer"(sb := #sb, mb_query := #mb_query);
END_FUNCTION_BLOCK

FUNCTION_BLOCK "Integron_OXY-DIOS-DSP"   // FB84, SCL
{ S7_Optimized_Access := 'TRUE' }
VERSION : 0.1
   VAR_INPUT
      mb_addr : USInt;
   END_VAR
   VAR_IN_OUT
      mb_query : "mb_query";
   END_VAR
   VAR
      sb : "mb_station_block_udt";
      read1 : Struct
         Sensor_status : Struct
            x08 : Bool;
            x09 : Bool;
            x10 : Bool;
            x11 : Bool;
            x12 : Bool;
            x13 : Bool;
            x14 : Bool;
            x15 : Bool;
            x00_Correct_indication : Bool;
            x01_Range_exceeded_error : Bool;
            x02_Measuring_window_status : Bool;   // (Must be replaced)
            x03_Cleaning : Bool;
            x04_Maintaining_values_after_cleaning : Bool;   // ("holding time") F= Real current value, T=Saved value
            x05_Output_short_circuit_OXYGEN_CONTROL : Bool;
            x06_Output_short_circuit_AIRBLAST_CLEANING : Bool;
            x07 : Bool;
         END_STRUCT;
         cO2_concentration : Real;   // [mg/L]
         sO2_saturation : Real;   // [%]
         Head_temperature : Real;   // [degree C]
         pO2_O2_partial_pressure : Real;   // [bar]
         Tau_fluorescence_decay_time : Real;   // [us]
         Atmospheric_pressure : Real;   // [bar] (hydrostatic)
         Relative_humidity_inside_the_sensor : Real;   // [%]
         Humidity_sensor_temperature : Real;   // [degree C]
         Salinity : Real;   // [ppt]
         Mainboard_temperature : Real;   // [degree C]
         Sensor_serial_number : Array[1..4] of Word;
         Date_and_time : UDInt;   // [s]
         Window_serial_number : UInt;
         Expected_date_of_exchange_measuring_window : UDInt;   // [s]
         Date_of_last_calibration : UDInt;   // [s]
         RTC_battery_level : UInt;   // [%]
         Supply_power_24V : Real;
      END_STRUCT;
   END_VAR
BEGIN
   // Integron Poland EU - OXY-DIOS-DSP
   // Optical dissolved oxygen sensor
   // 
   // https://www.tme.eu/en/Document/9d0bf7a4d6041739cc6d58df1cc838cb/OXY-DIOS-DSP-Manual-EN-v.1.33.pdf
   // http://www.sensor.integron.pl

   "mb_station_block_header"(sb := #sb, mb_query := #mb_query);
   #mb_query.mb_addr := #mb_addr;

   #mb_query.mode := #mb_query.c.mode.read;
   #mb_query(data_addr := 41000, data_ptr := #read1);

   "mb_station_block_footer"(sb := #sb, mb_query := #mb_query);
END_FUNCTION_BLOCK

FUNCTION_BLOCK "masibus_85XX"   // FB86, SCL
{ S7_Optimized_Access := 'TRUE' }
VERSION : 0.1
   VAR_INPUT
      mb_addr : USInt;
   END_VAR
   VAR_IN_OUT
      mb_query : "mb_query";
   END_VAR
   VAR
      sb : "mb_station_block_udt";
      read1 : Struct
         channel : Array[1..24] of Int;
         Ambient_PV : Int;
         digital_output_status : DWord;
         alarm : Array[1..2] of DWord;
         control_status : DWord;
         alarm_blink_status : Array[1..2] of DWord;
         alarm_LED_status : Array[1..2] of DWord;
      END_STRUCT;
      write1_labels : Array[1..24] of String[6];
      write2_input_type : Array[1..24] of USInt;
   END_VAR
BEGIN
   // Masibus - 85XX+
   // SCANNER / DAQ
   // REF NO: m83B/om/101
   // http://www.masibus.com/Pmanual/Data_Acquisition/
   // Enhanced_Multi-Channel_Scanners/85XX+_User_Manual

   "mb_station_block_header"(sb := #sb,
                             mb_query := #mb_query);
   #mb_query.mb_addr := #mb_addr; // Device address.

   #mb_query.mode := #mb_query.c.mode.read;
   #mb_query(data_addr := 30001,
             data_ptr := #read1);

   #mb_query.mode := #mb_query.c.mode.write;
   #mb_query(data_addr := 42204,
             data_ptr := #write1_labels);
   #mb_query(data_addr := 40097,
             data_ptr := #write2_input_type);

   "mb_station_block_footer"(sb := #sb,
                             mb_query := #mb_query);

   (*

   #  : Type
   ------------
   00 : None
   01 : E-tc
   02 : J-tc
   03 : K-tc
   04 : T-tc
   05 : B-tc
   06 : R-tc 
   07 : S-tc
   08 : n-tc
   09 : RDT
   10 : Cu53
   11 : Ni120
   12 : -10.20mV
   13 : 0-100mV
   14 : 4-20mA
   15 : 0-20mA
   16 : 0-5V
   17 : 1-5V
   18 : 0-10V
   19 : Dig.inp

   *)
END_FUNCTION_BLOCK

